Yaskawa INFORM job: A_ROOF_UPPER_0614_2_PAINT_50.JBI

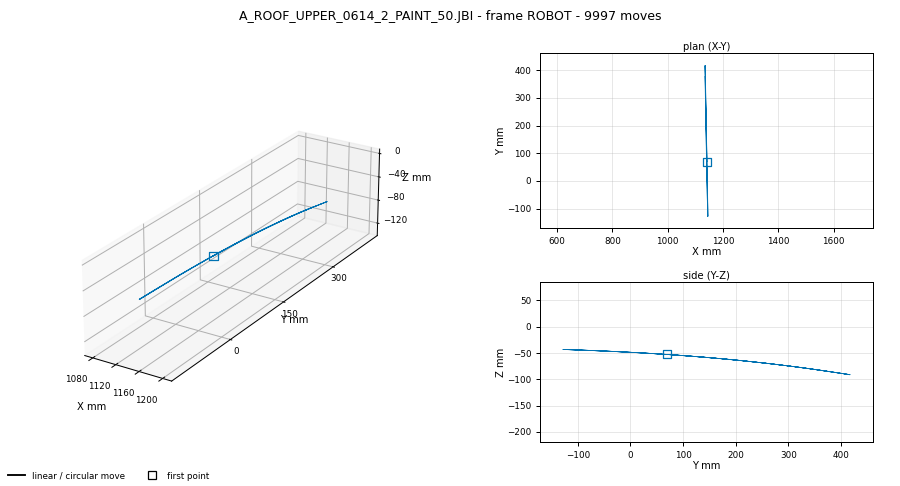
[picture p0: tool path of A_ROOF_UPPER_0614_2_PAINT_50.JBI in frame ROBOT, 9997 of 9997 moves have a stored position in this frame; points joined in program order, loops and branches not executed]
/JOB
//NAME A_ROOF_UPPER_0614_2_PAINT50
//POS
///NPOS 9997,0,0,0,0,0
///TOOL 1
///USER 0
///POSTYPE ROBOT
///RECTAN
///RCONF 1,0,0,0,0,0,0,0,0,0,0,0,0,0,0,0,0,0,0,0,0,0,0,0
C00000=1142.338,69.262,-52.629,-179.610,6.508,149.074
C00001=1142.333,69.511,-52.645,-179.607,6.509,149.073
C00002=1142.328,69.760,-52.662,-179.604,6.511,149.073
C00003=1142.323,70.010,-52.679,-179.601,6.511,149.072
C00004=1142.318,70.259,-52.695,-179.599,6.513,149.072
C00005=1142.313,70.509,-52.711,-179.596,6.515,149.071
C00006=1142.309,70.758,-52.728,-179.593,6.515,149.071
C00007=1142.303,71.007,-52.745,-179.591,6.517,149.070
C00008=1142.298,71.257,-52.762,-179.588,6.518,149.070
C00009=1142.294,71.506,-52.778,-179.585,6.519,149.069
C00010=1142.288,71.755,-52.795,-179.582,6.521,149.069
C00011=1142.284,72.005,-52.812,-179.580,6.522,149.068
C00012=1142.279,72.254,-52.828,-179.578,6.523,149.068
C00013=1142.273,72.503,-52.845,-179.574,6.524,149.067
C00014=1142.269,72.753,-52.862,-179.572,6.526,149.067
C00015=1142.264,73.003,-52.879,-179.569,6.527,149.066
C00016=1142.259,73.251,-52.896,-179.566,6.528,149.066
C00017=1142.254,73.501,-52.912,-179.563,6.530,149.065
C00018=1142.249,73.751,-52.930,-179.561,6.531,149.065
C00019=1142.244,74.000,-52.946,-179.559,6.532,149.064
C00020=1142.239,74.249,-52.962,-179.555,6.534,149.064
C00021=1142.234,74.499,-52.980,-179.553,6.535,149.063
C00022=1142.230,74.748,-52.996,-179.550,6.536,149.063
C00023=1142.224,74.997,-53.013,-179.548,6.538,149.062
C00024=1142.219,75.247,-53.030,-179.544,6.539,149.062
C00025=1142.214,75.497,-53.047,-179.542,6.540,149.061
C00026=1142.209,75.745,-53.064,-179.540,6.542,149.061
C00027=1142.205,75.995,-53.080,-179.537,6.543,149.060
C00028=1142.199,76.245,-53.097,-179.534,6.544,149.060
C00029=1142.195,76.494,-53.114,-179.531,6.546,149.059
C00030=1142.189,76.743,-53.132,-179.529,6.547,149.059
C00031=1142.185,76.992,-53.148,-179.526,6.548,149.058
C00032=1142.180,77.242,-53.166,-179.523,6.549,149.058
C00033=1142.175,77.491,-53.182,-179.521,6.551,149.057
C00034=1142.169,77.741,-53.199,-179.518,6.553,149.057
C00035=1142.165,77.990,-53.216,-179.515,6.553,149.056
C00036=1142.160,78.240,-53.233,-179.513,6.555,149.056
C00037=1142.155,78.489,-53.251,-179.510,6.556,149.055
C00038=1142.150,78.738,-53.268,-179.507,6.558,149.055
C00039=1142.145,78.987,-53.284,-179.504,6.559,149.054
C00040=1142.140,79.256,-53.303,-179.502,6.560,149.054
C00041=1142.134,79.525,-53.322,-179.499,6.562,149.054
C00042=1142.129,79.793,-53.339,-179.496,6.563,149.053
C00043=1142.124,80.061,-53.359,-179.493,6.565,149.052
C00044=1142.120,80.311,-53.375,-179.490,6.566,149.052
C00045=1142.114,80.560,-53.392,-179.487,6.568,149.051
C00046=1142.109,80.810,-53.410,-179.485,6.569,149.051
C00047=1142.104,81.058,-53.427,-179.482,6.570,149.051
C00048=1142.099,81.308,-53.444,-179.479,6.572,149.050
C00049=1142.095,81.558,-53.461,-179.476,6.573,149.049
C00050=1142.090,81.807,-53.479,-179.474,6.574,149.049
C00051=1142.084,82.056,-53.496,-179.471,6.576,149.049
C00052=1142.079,82.305,-53.512,-179.468,6.578,149.048
C00053=1142.075,82.555,-53.530,-179.465,6.579,149.048
C00054=1142.069,82.804,-53.548,-179.463,6.580,149.047
C00055=1142.065,83.054,-53.564,-179.460,6.581,149.047
C00056=1142.060,83.303,-53.582,-179.458,6.583,149.046
C00057=1142.055,83.553,-53.599,-179.454,6.584,149.046
C00058=1142.050,83.801,-53.617,-179.452,6.585,149.045
C00059=1142.045,84.051,-53.634,-179.450,6.587,149.045
C00060=1142.040,84.300,-53.652,-179.447,6.589,149.044
C00061=1142.035,84.549,-53.668,-179.444,6.590,149.044
C00062=1142.030,84.799,-53.686,-179.441,6.591,149.043
C00063=1142.025,85.048,-53.704,-179.439,6.592,149.043
C00064=1142.021,85.298,-53.720,-179.436,6.594,149.042
C00065=1142.016,85.547,-53.738,-179.433,6.596,149.042
C00066=1142.011,85.797,-53.756,-179.430,6.597,149.041
C00067=1142.006,86.046,-53.773,-179.428,6.598,149.041
C00068=1142.001,86.296,-53.790,-179.425,6.599,149.040
C00069=1141.996,86.544,-53.808,-179.422,6.601,149.040
C00070=1141.990,86.794,-53.825,-179.419,6.602,149.039
C00071=1141.986,87.043,-53.843,-179.417,6.603,149.039
C00072=1141.981,87.292,-53.861,-179.414,6.605,149.039
C00073=1141.976,87.542,-53.878,-179.411,6.607,149.038
C00074=1141.971,87.791,-53.896,-179.409,6.608,149.038
C00075=1141.966,88.041,-53.913,-179.406,6.610,149.037
C00076=1141.962,88.289,-53.930,-179.403,6.611,149.037
C00077=1141.957,88.539,-53.948,-179.401,6.612,149.036
C00078=1141.952,88.788,-53.966,-179.398,6.614,149.036
C00079=1141.947,89.038,-53.984,-179.395,6.615,149.035
C00080=1141.942,89.287,-54.001,-179.392,6.617,149.035
C00081=1141.937,89.537,-54.019,-179.390,6.618,149.034
C00082=1141.932,89.785,-54.036,-179.387,6.619,149.034
C00083=1141.927,90.035,-54.054,-179.384,6.621,149.033
C00084=1141.922,90.284,-54.072,-179.381,6.622,149.033
C00085=1141.917,90.534,-54.089,-179.378,6.624,149.032
C00086=1141.913,90.783,-54.107,-179.376,6.626,149.032
C00087=1141.907,91.033,-54.125,-179.373,6.627,149.032
C00088=1141.902,91.282,-54.143,-179.371,6.628,149.031
C00089=1141.898,91.531,-54.160,-179.368,6.630,149.030
C00090=1141.893,91.780,-54.178,-179.365,6.631,149.030
C00091=1141.888,92.030,-54.195,-179.362,6.633,149.030
C00092=1141.883,92.279,-54.213,-179.360,6.634,149.029
C00093=1141.878,92.528,-54.231,-179.357,6.635,149.029
C00094=1141.873,92.777,-54.249,-179.354,6.637,149.028
C00095=1141.868,93.027,-54.267,-179.351,6.638,149.028
C00096=1141.863,93.276,-54.285,-179.348,6.640,149.027
C00097=1141.858,93.525,-54.303,-179.346,6.642,149.027
C00098=1141.854,93.775,-54.321,-179.344,6.643,149.026
C00099=1141.849,94.024,-54.339,-179.340,6.644,149.026
C00100=1141.844,94.273,-54.357,-179.338,6.646,149.025
C00101=1141.839,94.523,-54.374,-179.335,6.647,149.025
C00102=1141.834,94.772,-54.392,-179.332,6.649,149.025
C00103=1141.829,95.022,-54.410,-179.329,6.651,149.024
C00104=1141.824,95.271,-54.428,-179.327,6.652,149.024
C00105=1141.819,95.520,-54.446,-179.324,6.653,149.023
C00106=1141.814,95.769,-54.464,-179.321,6.654,149.023
C00107=1141.809,96.018,-54.482,-179.319,6.656,149.022
C00108=1141.805,96.268,-54.500,-179.316,6.658,149.022
C00109=1141.800,96.517,-54.518,-179.313,6.659,149.021
C00110=1141.795,96.767,-54.536,-179.310,6.661,149.021
C00111=1141.790,97.016,-54.554,-179.307,6.662,149.020
C00112=1141.786,97.265,-54.572,-179.305,6.663,149.020
C00113=1141.781,97.514,-54.590,-179.302,6.665,149.020
C00114=1141.776,97.763,-54.608,-179.300,6.667,149.019
C00115=1141.771,98.012,-54.626,-179.297,6.668,149.019
C00116=1141.766,98.262,-54.645,-179.294,6.670,149.018
C00117=1141.762,98.511,-54.662,-179.291,6.671,149.018
C00118=1141.756,98.761,-54.681,-179.288,6.673,149.017
C00119=1141.751,99.010,-54.699,-179.285,6.675,149.017
C00120=1141.746,99.259,-54.717,-179.283,6.676,149.016
C00121=1141.741,99.509,-54.735,-179.281,6.677,149.016
C00122=1141.737,99.758,-54.753,-179.278,6.679,149.016
C00123=1141.732,100.008,-54.771,-179.275,6.680,149.015
C00124=1141.727,100.257,-54.789,-179.272,6.682,149.014
C00125=1141.722,100.506,-54.807,-179.269,6.684,149.014
C00126=1141.717,100.755,-54.827,-179.266,6.685,149.014
C00127=1141.712,101.005,-54.845,-179.264,6.687,149.013
C00128=1141.708,101.254,-54.863,-179.261,6.689,149.013
C00129=1141.703,101.503,-54.881,-179.258,6.689,149.012
C00130=1141.698,101.752,-54.899,-179.256,6.691,149.012
C00131=1141.692,102.002,-54.917,-179.253,6.692,149.011
C00132=1141.688,102.251,-54.936,-179.250,6.694,149.011
C00133=1141.683,102.500,-54.954,-179.247,6.696,149.011
C00134=1141.678,102.749,-54.972,-179.245,6.698,149.010
C00135=1141.673,102.998,-54.990,-179.242,6.699,149.010
C00136=1141.669,103.248,-55.010,-179.239,6.701,149.009
C00137=1141.664,103.497,-55.028,-179.236,6.702,149.009
C00138=1141.659,103.746,-55.046,-179.233,6.704,149.008
C00139=1141.654,103.996,-55.064,-179.231,6.706,149.008
C00140=1141.649,104.245,-55.084,-179.228,6.706,149.007
C00141=1141.644,104.494,-55.102,-179.226,6.708,149.007
C00142=1141.639,104.743,-55.120,-179.223,6.710,149.007
C00143=1141.635,104.993,-55.139,-179.220,6.711,149.006
C00144=1141.629,105.261,-55.159,-179.217,6.713,149.006
C00145=1141.624,105.530,-55.178,-179.214,6.715,149.005
C00146=1141.619,105.798,-55.198,-179.211,6.717,149.005
C00147=1141.614,106.066,-55.218,-179.208,6.718,149.004
C00148=1141.609,106.316,-55.237,-179.205,6.720,149.004
C00149=1141.604,106.565,-55.255,-179.202,6.722,149.003
C00150=1141.599,106.814,-55.274,-179.199,6.723,149.003
C00151=1141.594,107.064,-55.293,-179.197,6.725,149.002
C00152=1141.590,107.312,-55.312,-179.194,6.727,149.002
C00153=1141.584,107.562,-55.330,-179.192,6.728,149.002
C00154=1141.580,107.812,-55.348,-179.189,6.729,149.001
C00155=1141.575,108.060,-55.367,-179.186,6.731,149.001
C00156=1141.569,108.310,-55.386,-179.183,6.732,149.000
C00157=1141.565,108.559,-55.405,-179.180,6.734,149.000
C00158=1141.560,108.808,-55.423,-179.178,6.736,148.999
C00159=1141.555,109.057,-55.442,-179.175,6.737,148.999
C00160=1141.551,109.307,-55.460,-179.172,6.739,148.999
C00161=1141.545,109.556,-55.480,-179.170,6.741,148.998
C00162=1141.541,109.806,-55.498,-179.167,6.742,148.998
C00163=1141.536,110.055,-55.517,-179.164,6.744,148.997
C00164=1141.531,110.304,-55.535,-179.161,6.745,148.997
C00165=1141.527,110.553,-55.554,-179.158,6.747,148.996
C00166=1141.522,110.802,-55.574,-179.155,6.749,148.996
C00167=1141.517,111.052,-55.592,-179.153,6.750,148.995
C00168=1141.512,111.301,-55.611,-179.150,6.752,148.995
C00169=1141.507,111.550,-55.629,-179.147,6.754,148.995
C00170=1141.502,111.799,-55.649,-179.145,6.755,148.994
C00171=1141.498,112.048,-55.668,-179.142,6.757,148.994
C00172=1141.493,112.298,-55.687,-179.139,6.759,148.993
C00173=1141.488,112.547,-55.705,-179.136,6.760,148.993
C00174=1141.482,112.796,-55.724,-179.133,6.762,148.992
C00175=1141.478,113.046,-55.743,-179.130,6.764,148.992
C00176=1141.473,113.294,-55.762,-179.128,6.765,148.992
C00177=1141.468,113.544,-55.782,-179.125,6.767,148.991
C00178=1141.463,113.793,-55.800,-179.122,6.769,148.991
C00179=1141.459,114.043,-55.819,-179.119,6.770,148.990
C00180=1141.454,114.291,-55.838,-179.117,6.772,148.990
C00181=1141.449,114.541,-55.857,-179.114,6.774,148.990
C00182=1141.444,114.790,-55.876,-179.111,6.775,148.989
C00183=1141.440,115.039,-55.895,-179.109,6.777,148.989
C00184=1141.434,115.288,-55.915,-179.106,6.779,148.988
C00185=1141.430,115.538,-55.933,-179.103,6.780,148.988
C00186=1141.425,115.787,-55.952,-179.100,6.782,148.987
C00187=1141.420,116.037,-55.972,-179.097,6.783,148.987
C00188=1141.415,116.285,-55.991,-179.094,6.785,148.986
C00189=1141.410,116.535,-56.010,-179.092,6.787,148.986
C00190=1141.406,116.783,-56.029,-179.089,6.788,148.986
C00191=1141.401,117.034,-56.048,-179.086,6.790,148.985
C00192=1141.395,117.282,-56.067,-179.084,6.792,148.985
C00193=1141.391,117.532,-56.086,-179.081,6.794,148.984
C00194=1141.386,117.781,-56.106,-179.078,6.795,148.984
C00195=1141.381,118.030,-56.125,-179.075,6.797,148.984
C00196=1141.376,118.279,-56.145,-179.073,6.799,148.983
C00197=1141.372,118.528,-56.164,-179.070,6.800,148.983
C00198=1141.367,118.777,-56.183,-179.067,6.802,148.982
C00199=1141.362,119.027,-56.203,-179.064,6.804,148.982
C00200=1141.357,119.276,-56.221,-179.062,6.805,148.982
C00201=1141.352,119.525,-56.240,-179.059,6.807,148.981
C00202=1141.348,119.775,-56.260,-179.056,6.808,148.981
C00203=1141.342,120.024,-56.279,-179.053,6.810,148.980
C00204=1141.338,120.273,-56.298,-179.050,6.812,148.980
C00205=1141.333,120.522,-56.318,-179.048,6.813,148.979
C00206=1141.328,120.772,-56.337,-179.045,6.815,148.979
C00207=1141.323,121.021,-56.357,-179.042,6.817,148.979
C00208=1141.319,121.270,-56.376,-179.039,6.819,148.978
C00209=1141.314,121.519,-56.396,-179.037,6.820,148.978
C00210=1141.309,121.767,-56.415,-179.034,6.822,148.977
C00211=1141.304,122.017,-56.435,-179.031,6.824,148.977
C00212=1141.299,122.267,-56.455,-179.028,6.826,148.977
C00213=1141.295,122.515,-56.473,-179.025,6.828,148.976
C00214=1141.290,122.765,-56.493,-179.023,6.830,148.976
C00215=1141.285,123.014,-56.513,-179.020,6.831,148.975
C00216=1141.280,123.263,-56.532,-179.017,6.833,148.975
C00217=1141.275,123.513,-56.551,-179.014,6.835,148.975
C00218=1141.270,123.762,-56.571,-179.012,6.836,148.974
C00219=1141.266,124.010,-56.591,-179.009,6.838,148.974
C00220=1141.262,124.260,-56.610,-179.006,6.840,148.973
C00221=1141.256,124.509,-56.629,-179.003,6.841,148.973
C00222=1141.251,124.758,-56.649,-179.001,6.843,148.973
C00223=1141.247,125.008,-56.669,-178.998,6.845,148.972
C00224=1141.242,125.257,-56.689,-178.995,6.846,148.972
C00225=1141.237,125.506,-56.708,-178.992,6.849,148.971
C00226=1141.232,125.755,-56.728,-178.989,6.851,148.971
C00227=1141.227,126.005,-56.748,-178.987,6.852,148.971
C00228=1141.223,126.253,-56.767,-178.984,6.854,148.970
C00229=1141.218,126.502,-56.787,-178.981,6.856,148.970
C00230=1141.214,126.752,-56.807,-178.978,6.857,148.969
C00231=1141.208,127.001,-56.826,-178.976,6.859,148.969
C00232=1141.204,127.250,-56.846,-178.973,6.861,148.969
C00233=1141.199,127.499,-56.866,-178.970,6.863,148.968
C00234=1141.194,127.749,-56.885,-178.967,6.864,148.968
C00235=1141.189,127.997,-56.905,-178.965,6.866,148.967
C00236=1141.185,128.247,-56.925,-178.961,6.868,148.967
C00237=1141.180,128.496,-56.945,-178.959,6.870,148.967
C00238=1141.175,128.745,-56.965,-178.956,6.872,148.966
C00239=1141.170,128.994,-56.984,-178.953,6.873,148.966
C00240=1141.166,129.243,-57.005,-178.951,6.875,148.965
C00241=1141.161,129.493,-57.024,-178.948,6.877,148.965
C00242=1141.156,129.742,-57.044,-178.945,6.879,148.965
C00243=1141.151,129.990,-57.064,-178.942,6.880,148.964
C00244=1141.146,130.240,-57.084,-178.940,6.882,148.964
C00245=1141.141,130.489,-57.105,-178.936,6.884,148.963
C00246=1141.136,130.739,-57.124,-178.934,6.886,148.963
C00247=1141.132,130.988,-57.145,-178.931,6.888,148.963
C00248=1141.127,131.256,-57.166,-178.928,6.890,148.962
C00249=1141.121,131.525,-57.188,-178.925,6.892,148.962
C00250=1141.117,131.793,-57.209,-178.922,6.893,148.961
C00251=1141.111,132.061,-57.230,-178.919,6.895,148.961
C00252=1141.106,132.311,-57.251,-178.916,6.897,148.960
C00253=1141.101,132.560,-57.271,-178.913,6.899,148.960
C00254=1141.097,132.809,-57.291,-178.910,6.901,148.960
C00255=1141.092,133.059,-57.311,-178.908,6.903,148.959
C00256=1141.088,133.308,-57.331,-178.905,6.904,148.959
C00257=1141.082,133.556,-57.350,-178.903,6.906,148.959
C00258=1141.077,133.806,-57.371,-178.900,6.908,148.958
C00259=1141.073,134.055,-57.392,-178.897,6.910,148.958
C00260=1141.068,134.304,-57.411,-178.894,6.912,148.958
C00261=1141.064,134.553,-57.432,-178.891,6.914,148.957
C00262=1141.059,134.802,-57.452,-178.888,6.916,148.957
C00263=1141.054,135.052,-57.472,-178.886,6.917,148.956
C00264=1141.049,135.301,-57.493,-178.883,6.919,148.956
C00265=1141.044,135.549,-57.513,-178.880,6.921,148.956
C00266=1141.040,135.799,-57.532,-178.877,6.923,148.955
C00267=1141.035,136.048,-57.553,-178.874,6.925,148.955
C00268=1141.030,136.297,-57.574,-178.871,6.927,148.954
C00269=1141.025,136.547,-57.593,-178.869,6.929,148.954
C00270=1141.021,136.795,-57.614,-178.866,6.930,148.954
C00271=1141.016,137.044,-57.634,-178.863,6.932,148.953
C00272=1141.011,137.294,-57.655,-178.860,6.934,148.953
C00273=1141.006,137.543,-57.675,-178.857,6.936,148.952
C00274=1141.002,137.792,-57.695,-178.855,6.938,148.952
C00275=1140.997,138.041,-57.716,-178.852,6.940,148.952
C00276=1140.992,138.290,-57.736,-178.850,6.942,148.952
C00277=1140.988,138.539,-57.757,-178.846,6.944,148.951
C00278=1140.982,138.788,-57.777,-178.844,6.946,148.951
C00279=1140.977,139.037,-57.797,-178.841,6.948,148.950
C00280=1140.973,139.286,-57.817,-178.838,6.949,148.950
C00281=1140.968,139.536,-57.838,-178.835,6.951,148.950
C00282=1140.963,139.785,-57.859,-178.833,6.953,148.949
C00283=1140.959,140.034,-57.879,-178.829,6.955,148.949
C00284=1140.954,140.283,-57.900,-178.827,6.957,148.948
C00285=1140.949,140.532,-57.921,-178.824,6.959,148.948
C00286=1140.945,140.781,-57.941,-178.821,6.960,148.948
C00287=1140.940,141.030,-57.962,-178.819,6.962,148.947
C00288=1140.935,141.279,-57.982,-178.816,6.965,148.947
C00289=1140.930,141.528,-58.003,-178.813,6.967,148.947
C00290=1140.926,141.777,-58.024,-178.810,6.968,148.946
C00291=1140.921,142.026,-58.044,-178.808,6.970,148.946
C00292=1140.916,142.275,-58.065,-178.804,6.972,148.946
C00293=1140.912,142.524,-58.085,-178.802,6.974,148.945
C00294=1140.907,142.774,-58.107,-178.799,6.976,148.945
C00295=1140.903,143.023,-58.127,-178.796,6.978,148.944
C00296=1140.897,143.272,-58.148,-178.793,6.979,148.944
C00297=1140.893,143.521,-58.168,-178.790,6.982,148.944
C00298=1140.888,143.771,-58.189,-178.788,6.984,148.943
C00299=1140.883,144.020,-58.210,-178.785,6.986,148.943
C00300=1140.879,144.269,-58.230,-178.782,6.987,148.943
C00301=1140.874,144.518,-58.251,-178.779,6.990,148.942
C00302=1140.869,144.767,-58.271,-178.776,6.991,148.942
C00303=1140.864,145.016,-58.292,-178.774,6.993,148.942
C00304=1140.859,145.265,-58.313,-178.771,6.995,148.941
C00305=1140.855,145.514,-58.334,-178.768,6.997,148.941
C00306=1140.850,145.763,-58.355,-178.765,6.999,148.940
C00307=1140.845,146.012,-58.376,-178.763,7.001,148.940
C00308=1140.841,146.262,-58.397,-178.760,7.003,148.940
C00309=1140.836,146.511,-58.417,-178.757,7.005,148.939
C00310=1140.831,146.759,-58.439,-178.754,7.007,148.939
C00311=1140.827,147.008,-58.460,-178.751,7.009,148.939
C00312=1140.822,147.258,-58.480,-178.749,7.011,148.938
C00313=1140.817,147.507,-58.501,-178.746,7.012,148.938
C00314=1140.812,147.756,-58.522,-178.743,7.015,148.938
C00315=1140.807,148.004,-58.544,-178.740,7.017,148.937
C00316=1140.803,148.254,-58.565,-178.738,7.019,148.937
C00317=1140.798,148.503,-58.585,-178.734,7.021,148.937
C00318=1140.793,148.752,-58.607,-178.732,7.023,148.936
C00319=1140.789,149.001,-58.627,-178.729,7.024,148.936
C00320=1140.784,149.250,-58.648,-178.726,7.026,148.935
C00321=1140.779,149.499,-58.670,-178.723,7.029,148.935
C00322=1140.775,149.749,-58.691,-178.721,7.031,148.935
C00323=1140.770,149.998,-58.712,-178.718,7.032,148.935
C00324=1140.765,150.246,-58.733,-178.715,7.034,148.934
C00325=1140.760,150.496,-58.754,-178.712,7.037,148.934
C00326=1140.755,150.745,-58.775,-178.709,7.038,148.933
C00327=1140.751,150.994,-58.797,-178.707,7.040,148.933
C00328=1140.746,151.243,-58.818,-178.704,7.043,148.933
C00329=1140.742,151.492,-58.839,-178.701,7.045,148.933
C00330=1140.737,151.741,-58.860,-178.698,7.046,148.932
C00331=1140.732,151.989,-58.881,-178.695,7.048,148.932
C00332=1140.727,152.239,-58.903,-178.692,7.051,148.931
C00333=1140.723,152.488,-58.924,-178.690,7.053,148.931
C00334=1140.718,152.737,-58.945,-178.687,7.054,148.931
C00335=1140.713,152.986,-58.966,-178.684,7.057,148.930
C00336=1140.708,153.236,-58.988,-178.681,7.059,148.930
C00337=1140.704,153.484,-59.009,-178.678,7.060,148.930
C00338=1140.699,153.733,-59.030,-178.675,7.063,148.929
C00339=1140.694,153.982,-59.052,-178.673,7.065,148.929
C00340=1140.690,154.232,-59.073,-178.670,7.067,148.929
C00341=1140.685,154.480,-59.095,-178.668,7.068,148.928
C00342=1140.680,154.730,-59.116,-178.664,7.071,148.928
C00343=1140.675,154.978,-59.137,-178.662,7.073,148.928
C00344=1140.671,155.227,-59.159,-178.659,7.075,148.928
C00345=1140.666,155.477,-59.180,-178.656,7.077,148.927
C00346=1140.661,155.725,-59.201,-178.653,7.079,148.927
C00347=1140.657,155.975,-59.223,-178.651,7.081,148.926
C00348=1140.652,156.224,-59.244,-178.647,7.083,148.926
C00349=1140.647,156.472,-59.266,-178.645,7.085,148.926
C00350=1140.643,156.722,-59.288,-178.642,7.087,148.925
C00351=1140.637,156.971,-59.309,-178.639,7.090,148.925
C00352=1140.633,157.240,-59.332,-178.636,7.091,148.925
C00353=1140.627,157.509,-59.356,-178.633,7.094,148.924
C00354=1140.623,157.778,-59.379,-178.630,7.095,148.924
C00355=1140.618,158.047,-59.403,-178.627,7.098,148.924
C00356=1140.612,158.296,-59.424,-178.625,7.100,148.923
C00357=1140.608,158.545,-59.445,-178.621,7.103,148.923
C00358=1140.604,158.794,-59.467,-178.619,7.104,148.923
C00359=1140.599,159.042,-59.488,-178.616,7.106,148.922
C00360=1140.594,159.291,-59.509,-178.613,7.109,148.922
C00361=1140.590,159.541,-59.531,-178.611,7.111,148.922
C00362=1140.585,159.789,-59.553,-178.607,7.113,148.921
C00363=1140.581,160.039,-59.575,-178.605,7.115,148.921
C00364=1140.576,160.287,-59.597,-178.602,7.117,148.921
C00365=1140.571,160.536,-59.619,-178.599,7.119,148.921
C00366=1140.567,160.785,-59.641,-178.596,7.121,148.920
C00367=1140.561,161.035,-59.662,-178.594,7.123,148.920
C00368=1140.556,161.284,-59.684,-178.590,7.125,148.919
C00369=1140.551,161.533,-59.706,-178.588,7.127,148.919
C00370=1140.547,161.782,-59.728,-178.585,7.129,148.919
C00371=1140.542,162.031,-59.750,-178.582,7.132,148.919
C00372=1140.537,162.280,-59.771,-178.579,7.133,148.918
C00373=1140.533,162.529,-59.793,-178.577,7.136,148.918
C00374=1140.528,162.778,-59.815,-178.574,7.138,148.918
C00375=1140.524,163.027,-59.837,-178.571,7.140,148.917
C00376=1140.519,163.276,-59.859,-178.568,7.142,148.917
C00377=1140.515,163.525,-59.881,-178.566,7.144,148.917
C00378=1140.510,163.774,-59.903,-178.563,7.146,148.916
C00379=1140.506,164.023,-59.925,-178.560,7.149,148.916
C00380=1140.500,164.272,-59.947,-178.557,7.150,148.916
C00381=1140.496,164.521,-59.969,-178.554,7.153,148.916
C00382=1140.491,164.770,-59.991,-178.551,7.155,148.915
C00383=1140.487,165.019,-60.013,-178.549,7.157,148.915
C00384=1140.482,165.268,-60.034,-178.545,7.159,148.914
C00385=1140.478,165.517,-60.057,-178.543,7.161,148.914
C00386=1140.472,165.765,-60.079,-178.540,7.164,148.914
C00387=1140.468,166.015,-60.101,-178.537,7.166,148.914
C00388=1140.463,166.263,-60.123,-178.535,7.168,148.913
C00389=1140.459,166.513,-60.145,-178.532,7.170,148.913
C00390=1140.454,166.761,-60.167,-178.529,7.172,148.913
C00391=1140.449,167.011,-60.189,-178.526,7.174,148.912
C00392=1140.445,167.259,-60.212,-178.523,7.176,148.912
C00393=1140.440,167.508,-60.234,-178.521,7.178,148.912
C00394=1140.435,167.757,-60.256,-178.517,7.181,148.911
C00395=1140.430,168.007,-60.278,-178.515,7.183,148.911
C00396=1140.426,168.255,-60.301,-178.512,7.185,148.911
C00397=1140.422,168.504,-60.323,-178.509,7.187,148.911
C00398=1140.417,168.754,-60.345,-178.506,7.190,148.910
C00399=1140.412,169.002,-60.367,-178.504,7.192,148.910
C00400=1140.408,169.251,-60.390,-178.501,7.193,148.910
C00401=1140.403,169.500,-60.411,-178.498,7.196,148.909
C00402=1140.398,169.749,-60.434,-178.495,7.198,148.909
C00403=1140.394,169.998,-60.457,-178.492,7.200,148.909
C00404=1140.389,170.247,-60.479,-178.489,7.202,148.908
C00405=1140.384,170.496,-60.501,-178.487,7.205,148.908
C00406=1140.379,170.744,-60.524,-178.484,7.207,148.908
C00407=1140.374,170.994,-60.546,-178.481,7.209,148.908
C00408=1140.370,171.243,-60.568,-178.478,7.211,148.907
C00409=1140.366,171.491,-60.591,-178.476,7.213,148.907
C00410=1140.361,171.741,-60.613,-178.472,7.216,148.907
C00411=1140.356,171.989,-60.636,-178.470,7.218,148.907
C00412=1140.352,172.238,-60.658,-178.467,7.220,148.906
C00413=1140.347,172.488,-60.680,-178.464,7.222,148.906
C00414=1140.342,172.736,-60.703,-178.461,7.225,148.906
C00415=1140.337,172.986,-60.725,-178.459,7.227,148.905
C00416=1140.333,173.235,-60.748,-178.455,7.229,148.905
C00417=1140.328,173.483,-60.770,-178.453,7.231,148.905
C00418=1140.324,173.732,-60.793,-178.450,7.233,148.905
C00419=1140.319,173.982,-60.816,-178.447,7.235,148.904
C00420=1140.314,174.230,-60.838,-178.445,7.238,148.904
C00421=1140.310,174.479,-60.861,-178.442,7.240,148.904
C00422=1140.305,174.728,-60.884,-178.439,7.242,148.904
C00423=1140.301,174.977,-60.906,-178.436,7.245,148.903
C00424=1140.296,175.226,-60.929,-178.433,7.246,148.903
C00425=1140.292,175.475,-60.952,-178.430,7.249,148.903
C00426=1140.287,175.724,-60.974,-178.428,7.251,148.902
C00427=1140.282,175.972,-60.997,-178.425,7.254,148.902
C00428=1140.277,176.221,-61.020,-178.422,7.256,148.902
C00429=1140.272,176.471,-61.043,-178.419,7.258,148.901
C00430=1140.268,176.720,-61.065,-178.416,7.260,148.901
C00431=1140.263,176.968,-61.088,-178.413,7.263,148.901
C00432=1140.259,177.217,-61.110,-178.411,7.265,148.901
C00433=1140.254,177.466,-61.134,-178.408,7.267,148.900
C00434=1140.250,177.715,-61.156,-178.405,7.269,148.900
C00435=1140.245,177.964,-61.179,-178.402,7.272,148.900
C00436=1140.240,178.213,-61.202,-178.400,7.274,148.900
C00437=1140.236,178.462,-61.225,-178.396,7.276,148.899
C00438=1140.231,178.711,-61.248,-178.394,7.278,148.899
C00439=1140.226,178.960,-61.270,-178.391,7.281,148.899
C00440=1140.222,179.209,-61.293,-178.388,7.283,148.898
C00441=1140.217,179.458,-61.317,-178.385,7.286,148.898
C00442=1140.213,179.706,-61.339,-178.383,7.287,148.898
C00443=1140.208,179.955,-61.363,-178.380,7.290,148.898
C00444=1140.204,180.204,-61.386,-178.377,7.292,148.897
C00445=1140.199,180.453,-61.408,-178.374,7.294,148.897
C00446=1140.194,180.702,-61.431,-178.372,7.297,148.897
C00447=1140.189,180.951,-61.455,-178.368,7.299,148.897
C00448=1140.185,181.200,-61.477,-178.366,7.301,148.896
C00449=1140.181,181.449,-61.501,-178.363,7.304,148.896
C00450=1140.176,181.698,-61.524,-178.360,7.305,148.896
C00451=1140.171,181.946,-61.546,-178.357,7.308,148.896
C00452=1140.167,182.195,-61.570,-178.355,7.310,148.895
C00453=1140.162,182.444,-61.593,-178.352,7.313,148.895
C00454=1140.157,182.693,-61.616,-178.349,7.315,148.895
C00455=1140.153,182.942,-61.639,-178.346,7.318,148.895
C00456=1140.148,183.211,-61.664,-178.343,7.320,148.894
C00457=1140.143,183.481,-61.689,-178.340,7.323,148.894
C00458=1140.137,183.751,-61.714,-178.336,7.325,148.894
C00459=1140.133,184.020,-61.739,-178.334,7.327,148.893
C00460=1140.128,184.269,-61.762,-178.331,7.330,148.893
C00461=1140.124,184.518,-61.786,-178.328,7.333,148.893
C00462=1140.119,184.767,-61.810,-178.325,7.334,148.893
C00463=1140.114,185.016,-61.833,-178.323,7.337,148.893
C00464=1140.110,185.265,-61.856,-178.320,7.339,148.892
C00465=1140.106,185.514,-61.879,-178.317,7.342,148.892
C00466=1140.101,185.763,-61.902,-178.314,7.344,148.892
C00467=1140.096,186.012,-61.926,-178.311,7.346,148.891
C00468=1140.091,186.261,-61.949,-178.309,7.348,148.891
C00469=1140.087,186.510,-61.972,-178.306,7.351,148.891
C00470=1140.082,186.758,-61.997,-178.303,7.354,148.891
C00471=1140.078,187.007,-62.020,-178.300,7.355,148.890
C00472=1140.074,187.256,-62.043,-178.297,7.358,148.890
C00473=1140.069,187.505,-62.066,-178.295,7.360,148.890
C00474=1140.064,187.753,-62.089,-178.292,7.363,148.890
C00475=1140.059,188.002,-62.113,-178.289,7.365,148.889
C00476=1140.055,188.251,-62.136,-178.286,7.368,148.889
C00477=1140.050,188.500,-62.160,-178.283,7.370,148.889
C00478=1140.045,188.749,-62.183,-178.281,7.372,148.889
C00479=1140.041,188.997,-62.207,-178.277,7.375,148.889
C00480=1140.036,189.246,-62.231,-178.275,7.377,148.888
C00481=1140.031,189.495,-62.254,-178.272,7.379,148.888
C00482=1140.027,189.744,-62.277,-178.269,7.382,148.888
C00483=1140.022,189.993,-62.301,-178.266,7.384,148.888
C00484=1140.018,190.242,-62.325,-178.264,7.387,148.887
C00485=1140.013,190.491,-62.348,-178.261,7.389,148.887
C00486=1140.009,190.739,-62.372,-178.258,7.392,148.887
C00487=1140.004,190.989,-62.396,-178.255,7.394,148.887
C00488=1140.000,191.237,-62.420,-178.253,7.396,148.886
C00489=1139.995,191.486,-62.443,-178.249,7.399,148.886
C00490=1139.991,191.736,-62.467,-178.247,7.401,148.886
C00491=1139.986,191.984,-62.491,-178.244,7.403,148.886
C00492=1139.982,192.233,-62.514,-178.241,7.406,148.886
C00493=1139.977,192.481,-62.538,-178.238,7.408,148.885
C00494=1139.972,192.731,-62.562,-178.236,7.411,148.885
C00495=1139.967,192.979,-62.586,-178.233,7.413,148.885
C00496=1139.963,193.228,-62.610,-178.230,7.416,148.885
C00497=1139.958,193.477,-62.634,-178.227,7.418,148.884
C00498=1139.954,193.726,-62.657,-178.225,7.420,148.884
C00499=1139.949,193.974,-62.681,-178.221,7.423,148.884
C00500=1139.945,194.224,-62.705,-178.218,7.426,148.884
C00501=1139.941,194.472,-62.729,-178.216,7.427,148.883
C00502=1139.935,194.721,-62.753,-178.213,7.430,148.883
C00503=1139.931,194.970,-62.777,-178.211,7.432,148.883
C00504=1139.926,195.219,-62.800,-178.207,7.435,148.883
C00505=1139.922,195.467,-62.824,-178.205,7.438,148.883
C00506=1139.917,195.716,-62.848,-178.202,7.440,148.882
C00507=1139.913,195.965,-62.872,-178.199,7.442,148.882
C00508=1139.908,196.214,-62.897,-178.196,7.445,148.882
C00509=1139.904,196.463,-62.921,-178.194,7.447,148.882
C00510=1139.899,196.712,-62.944,-178.190,7.450,148.881
C00511=1139.895,196.960,-62.968,-178.188,7.452,148.881
C00512=1139.889,197.209,-62.993,-178.185,7.455,148.881
C00513=1139.885,197.458,-63.016,-178.182,7.457,148.881
C00514=1139.881,197.707,-63.041,-178.179,7.460,148.881
C00515=1139.877,197.955,-63.065,-178.177,7.462,148.880
C00516=1139.871,198.204,-63.090,-178.174,7.465,148.880
C00517=1139.867,198.453,-63.113,-178.170,7.467,148.880
C00518=1139.862,198.702,-63.137,-178.168,7.469,148.880
C00519=1139.859,198.951,-63.161,-178.165,7.472,148.880
C00520=1139.853,199.199,-63.186,-178.162,7.475,148.879
C00521=1139.849,199.448,-63.209,-178.160,7.477,148.879
C00522=1139.844,199.697,-63.234,-178.157,7.479,148.879
C00523=1139.840,199.946,-63.259,-178.154,7.482,148.879
C00524=1139.835,200.195,-63.283,-178.152,7.484,148.879
C00525=1139.831,200.443,-63.307,-178.148,7.487,148.878
C00526=1139.826,200.692,-63.331,-178.145,7.490,148.878
C00527=1139.822,200.941,-63.356,-178.143,7.492,148.878
C00528=1139.818,201.189,-63.380,-178.140,7.494,148.878
C00529=1139.812,201.439,-63.404,-178.137,7.497,148.878
C00530=1139.808,201.687,-63.428,-178.134,7.499,148.877
C00531=1139.803,201.936,-63.453,-178.132,7.502,148.877
C00532=1139.799,202.185,-63.477,-178.128,7.505,148.877
C00533=1139.795,202.433,-63.501,-178.126,7.507,148.877
C00534=1139.790,202.683,-63.526,-178.123,7.510,148.877
C00535=1139.786,202.931,-63.550,-178.120,7.512,148.876
C00536=1139.780,203.180,-63.575,-178.117,7.515,148.876
C00537=1139.776,203.428,-63.599,-178.115,7.517,148.876
C00538=1139.772,203.678,-63.624,-178.112,7.520,148.876
C00539=1139.767,203.926,-63.648,-178.109,7.523,148.876
C00540=1139.763,204.175,-63.672,-178.106,7.524,148.875
C00541=1139.758,204.424,-63.697,-178.103,7.527,148.875
C00542=1139.754,204.672,-63.721,-178.101,7.530,148.875
C00543=1139.749,204.920,-63.747,-178.097,7.533,148.875
C00544=1139.745,205.170,-63.771,-178.095,7.535,148.875
C00545=1139.740,205.418,-63.796,-178.092,7.538,148.874
C00546=1139.735,205.667,-63.820,-178.089,7.540,148.874
C00547=1139.731,205.916,-63.845,-178.087,7.542,148.874
C00548=1139.726,206.165,-63.870,-178.084,7.545,148.874
C00549=1139.722,206.414,-63.894,-178.081,7.548,148.874
C00550=1139.717,206.662,-63.919,-178.078,7.551,148.873
C00551=1139.713,206.910,-63.943,-178.076,7.553,148.873
C00552=1139.709,207.160,-63.968,-178.072,7.555,148.873
C00553=1139.703,207.409,-63.993,-178.070,7.558,148.873
C00554=1139.699,207.657,-64.017,-178.067,7.561,148.873
C00555=1139.695,207.906,-64.043,-178.064,7.563,148.872
C00556=1139.690,208.154,-64.067,-178.061,7.566,148.872
C00557=1139.686,208.404,-64.092,-178.059,7.569,148.872
C00558=1139.681,208.652,-64.117,-178.056,7.570,148.872
C00559=1139.677,208.900,-64.142,-178.053,7.573,148.872
C00560=1139.672,209.171,-64.169,-178.050,7.576,148.872
C00561=1139.667,209.442,-64.196,-178.047,7.579,148.871
C00562=1139.662,209.712,-64.223,-178.044,7.582,148.871
C00563=1139.657,209.983,-64.250,-178.040,7.585,148.871
C00564=1139.652,210.232,-64.275,-178.038,7.587,148.871
C00565=1139.648,210.481,-64.300,-178.035,7.590,148.871
C00566=1139.643,210.729,-64.325,-178.032,7.593,148.870
C00567=1139.639,210.979,-64.350,-178.029,7.595,148.870
C00568=1139.635,211.226,-64.374,-178.027,7.598,148.870
C00569=1139.630,211.476,-64.399,-178.024,7.600,148.870
C00570=1139.625,211.724,-64.425,-178.021,7.603,148.870
C00571=1139.621,211.973,-64.450,-178.018,7.606,148.870
C00572=1139.617,212.221,-64.475,-178.016,7.608,148.870
C00573=1139.612,212.471,-64.500,-178.013,7.611,148.869
C00574=1139.607,212.719,-64.525,-178.010,7.613,148.869
C00575=1139.603,212.968,-64.550,-178.007,7.616,148.869
C00576=1139.598,213.216,-64.576,-178.004,7.619,148.869
C00577=1139.594,213.465,-64.600,-178.001,7.621,148.869
C00578=1139.589,213.713,-64.625,-177.999,7.624,148.869
C00579=1139.585,213.963,-64.650,-177.996,7.627,148.868
C00580=1139.580,214.211,-64.676,-177.993,7.630,148.868
C00581=1139.576,214.460,-64.701,-177.990,7.632,148.868
C00582=1139.571,214.708,-64.726,-177.988,7.634,148.868
C00583=1139.567,214.957,-64.751,-177.985,7.637,148.868
C00584=1139.563,215.206,-64.776,-177.982,7.640,148.868
C00585=1139.558,215.455,-64.802,-177.979,7.643,148.867
C00586=1139.554,215.703,-64.827,-177.976,7.646,148.867
C00587=1139.548,215.952,-64.852,-177.974,7.648,148.867
C00588=1139.544,216.201,-64.878,-177.971,7.651,148.867
C00589=1139.539,216.449,-64.903,-177.968,7.653,148.867
C00590=1139.536,216.698,-64.928,-177.965,7.656,148.867
C00591=1139.531,216.947,-64.953,-177.962,7.659,148.867
C00592=1139.527,217.195,-64.979,-177.960,7.661,148.866
C00593=1139.522,217.444,-65.005,-177.957,7.664,148.866
C00594=1139.518,217.693,-65.030,-177.954,7.667,148.866
C00595=1139.513,217.941,-65.055,-177.951,7.669,148.866
C00596=1139.509,218.190,-65.081,-177.948,7.672,148.866
C00597=1139.504,218.438,-65.106,-177.946,7.674,148.866
C00598=1139.500,218.687,-65.132,-177.943,7.677,148.865
C00599=1139.495,218.937,-65.157,-177.940,7.680,148.865
C00600=1139.490,219.185,-65.182,-177.937,7.683,148.865
C00601=1139.486,219.433,-65.208,-177.934,7.686,148.865
C00602=1139.482,219.682,-65.234,-177.931,7.689,148.865
C00603=1139.477,219.930,-65.259,-177.929,7.690,148.865
C00604=1139.473,220.179,-65.285,-177.926,7.693,148.865
C00605=1139.469,220.428,-65.311,-177.923,7.696,148.864
C00606=1139.464,220.676,-65.336,-177.920,7.699,148.864
C00607=1139.459,220.925,-65.361,-177.917,7.702,148.864
C00608=1139.455,221.174,-65.387,-177.914,7.705,148.864
C00609=1139.451,221.423,-65.413,-177.912,7.707,148.864
C00610=1139.446,221.671,-65.438,-177.909,7.710,148.864
C00611=1139.442,221.920,-65.464,-177.906,7.713,148.864
C00612=1139.438,222.169,-65.490,-177.904,7.715,148.864
C00613=1139.432,222.417,-65.516,-177.901,7.718,148.863
C00614=1139.428,222.666,-65.541,-177.897,7.721,148.863
C00615=1139.424,222.915,-65.567,-177.895,7.724,148.863
C00616=1139.419,223.164,-65.593,-177.892,7.726,148.863
C00617=1139.415,223.411,-65.619,-177.890,7.729,148.863
C00618=1139.411,223.660,-65.645,-177.887,7.732,148.863
C00619=1139.406,223.909,-65.670,-177.884,7.735,148.863
C00620=1139.401,224.158,-65.697,-177.881,7.737,148.862
C00621=1139.397,224.406,-65.722,-177.878,7.740,148.862
C00622=1139.392,224.655,-65.748,-177.875,7.743,148.862
C00623=1139.388,224.904,-65.774,-177.872,7.746,148.862
C00624=1139.384,225.152,-65.799,-177.870,7.748,148.862
C00625=1139.379,225.400,-65.826,-177.867,7.751,148.862
C00626=1139.374,225.649,-65.852,-177.865,7.754,148.862
C00627=1139.370,225.898,-65.878,-177.861,7.756,148.861
C00628=1139.366,226.147,-65.903,-177.858,7.759,148.861
C00629=1139.362,226.395,-65.929,-177.856,7.762,148.861
C00630=1139.356,226.643,-65.956,-177.853,7.765,148.861
C00631=1139.352,226.892,-65.982,-177.850,7.768,148.861
C00632=1139.348,227.141,-66.007,-177.848,7.770,148.861
C00633=1139.343,227.390,-66.034,-177.845,7.773,148.861
C00634=1139.339,227.638,-66.060,-177.842,7.776,148.861
C00635=1139.335,227.887,-66.086,-177.839,7.778,148.861
C00636=1139.330,228.135,-66.111,-177.836,7.781,148.860
C00637=1139.325,228.383,-66.138,-177.833,7.784,148.860
C00638=1139.321,228.632,-66.164,-177.831,7.787,148.860
C00639=1139.317,228.881,-66.190,-177.828,7.790,148.860
C00640=1139.312,229.130,-66.217,-177.825,7.793,148.860
C00641=1139.308,229.378,-66.243,-177.822,7.796,148.860
C00642=1139.304,229.627,-66.268,-177.820,7.798,148.860
C00643=1139.299,229.875,-66.295,-177.817,7.801,148.860
C00644=1139.294,230.124,-66.321,-177.814,7.804,148.860
C00645=1139.290,230.372,-66.348,-177.811,7.806,148.859
C00646=1139.286,230.621,-66.374,-177.808,7.809,148.859
C00647=1139.282,230.869,-66.400,-177.805,7.812,148.859
C00648=1139.277,231.118,-66.426,-177.803,7.815,148.859
C00649=1139.273,231.367,-66.453,-177.800,7.818,148.859
C00650=1139.268,231.616,-66.479,-177.797,7.821,148.859
C00651=1139.264,231.864,-66.506,-177.794,7.824,148.859
C00652=1139.259,232.113,-66.532,-177.791,7.827,148.859
C00653=1139.255,232.361,-66.559,-177.789,7.829,148.859
C00654=1139.251,232.610,-66.584,-177.786,7.832,148.859
C00655=1139.246,232.858,-66.611,-177.784,7.835,148.858
C00656=1139.241,233.107,-66.637,-177.781,7.838,148.858
C00657=1139.237,233.355,-66.664,-177.778,7.840,148.858
C00658=1139.233,233.603,-66.690,-177.775,7.843,148.858
C00659=1139.228,233.852,-66.717,-177.772,7.846,148.858
C00660=1139.224,234.101,-66.743,-177.769,7.849,148.858
C00661=1139.219,234.349,-66.770,-177.766,7.852,148.858
C00662=1139.214,234.598,-66.796,-177.764,7.855,148.858
C00663=1139.210,234.846,-66.823,-177.761,7.858,148.858
C00664=1139.206,235.119,-66.853,-177.758,7.861,148.858
C00665=1139.200,235.391,-66.881,-177.755,7.863,148.857
C00666=1139.196,235.662,-66.910,-177.752,7.867,148.857
C00667=1139.191,235.934,-66.940,-177.749,7.870,148.857
C00668=1139.187,236.183,-66.967,-177.746,7.873,148.857
C00669=1139.183,236.432,-66.993,-177.743,7.876,148.857
C00670=1139.178,236.680,-67.020,-177.740,7.879,148.857
C00671=1139.174,236.928,-67.046,-177.737,7.881,148.857
C00672=1139.169,237.177,-67.073,-177.735,7.884,148.857
C00673=1139.164,237.426,-67.099,-177.732,7.887,148.857
C00674=1139.160,237.674,-67.126,-177.729,7.890,148.856
C00675=1139.156,237.923,-67.153,-177.726,7.893,148.856
C00676=1139.151,238.171,-67.180,-177.723,7.896,148.856
C00677=1139.147,238.419,-67.207,-177.721,7.899,148.856
C00678=1139.143,238.668,-67.234,-177.718,7.902,148.856
C00679=1139.138,238.916,-67.261,-177.715,7.905,148.856
C00680=1139.134,239.165,-67.287,-177.712,7.908,148.856
C00681=1139.129,239.413,-67.314,-177.709,7.911,148.856
C00682=1139.124,239.662,-67.341,-177.707,7.913,148.856
C00683=1139.120,239.911,-67.368,-177.704,7.916,148.856
C00684=1139.116,240.160,-67.394,-177.701,7.919,148.856
C00685=1139.112,240.408,-67.421,-177.698,7.922,148.856
C00686=1139.107,240.657,-67.449,-177.696,7.924,148.855
C00687=1139.102,240.905,-67.476,-177.693,7.927,148.855
C00688=1139.098,241.153,-67.502,-177.690,7.930,148.855
C00689=1139.094,241.402,-67.529,-177.688,7.933,148.855
C00690=1139.089,241.650,-67.557,-177.685,7.936,148.855
C00691=1139.085,241.899,-67.584,-177.682,7.939,148.855
C00692=1139.081,242.147,-67.611,-177.679,7.942,148.855
C00693=1139.077,242.395,-67.638,-177.676,7.945,148.855
C00694=1139.072,242.644,-67.665,-177.674,7.948,148.855
C00695=1139.067,242.892,-67.692,-177.671,7.951,148.855
C00696=1139.063,243.141,-67.719,-177.668,7.953,148.855
C00697=1139.059,243.390,-67.746,-177.665,7.956,148.855
C00698=1139.055,243.638,-67.773,-177.662,7.959,148.855
C00699=1139.051,243.886,-67.801,-177.660,7.963,148.855
C00700=1139.046,244.135,-67.828,-177.657,7.965,148.855
C00701=1139.041,244.383,-67.855,-177.654,7.968,148.855
C00702=1139.037,244.632,-67.882,-177.652,7.971,148.854
C00703=1139.032,244.881,-67.909,-177.649,7.974,148.854
C00704=1139.028,245.129,-67.937,-177.646,7.977,148.854
C00705=1139.023,245.377,-67.964,-177.643,7.980,148.854
C00706=1139.019,245.626,-67.992,-177.640,7.983,148.854
C00707=1139.015,245.875,-68.019,-177.637,7.987,148.854
C00708=1139.010,246.123,-68.046,-177.634,7.990,148.854
C00709=1139.006,246.371,-68.073,-177.631,7.992,148.854
C00710=1139.002,246.620,-68.100,-177.629,7.995,148.854
C00711=1138.998,246.868,-68.128,-177.626,7.998,148.854
C00712=1138.993,247.117,-68.155,-177.623,8.001,148.854
C00713=1138.989,247.365,-68.182,-177.620,8.004,148.854
C00714=1138.985,247.614,-68.210,-177.617,8.007,148.854
C00715=1138.980,247.862,-68.237,-177.615,8.010,148.854
C00716=1138.976,248.110,-68.265,-177.612,8.013,148.853
C00717=1138.971,248.359,-68.292,-177.609,8.016,148.854
C00718=1138.967,248.608,-68.320,-177.607,8.019,148.854
C00719=1138.962,248.856,-68.348,-177.604,8.022,148.853
C00720=1138.958,249.104,-68.375,-177.601,8.025,148.853
C00721=1138.954,249.353,-68.403,-177.598,8.028,148.853
C00722=1138.949,249.602,-68.430,-177.595,8.031,148.853
C00723=1138.945,249.849,-68.458,-177.593,8.034,148.853
C00724=1138.941,250.099,-68.486,-177.590,8.037,148.853
C00725=1138.936,250.346,-68.513,-177.587,8.039,148.853
C00726=1138.932,250.595,-68.540,-177.584,8.042,148.853
C00727=1138.928,250.844,-68.569,-177.582,8.045,148.853
C00728=1138.924,251.091,-68.596,-177.579,8.049,148.853
C00729=1138.919,251.340,-68.623,-177.576,8.051,148.853
C00730=1138.914,251.589,-68.652,-177.574,8.054,148.853
C00731=1138.910,251.837,-68.679,-177.571,8.057,148.853
C00732=1138.905,252.085,-68.707,-177.567,8.061,148.853
C00733=1138.902,252.334,-68.735,-177.565,8.064,148.853
C00734=1138.897,252.582,-68.762,-177.562,8.067,148.853
C00735=1138.893,252.831,-68.790,-177.559,8.070,148.853
C00736=1138.888,253.079,-68.819,-177.557,8.073,148.853
C00737=1138.884,253.327,-68.846,-177.554,8.076,148.853
C00738=1138.880,253.576,-68.874,-177.551,8.079,148.853
C00739=1138.875,253.824,-68.902,-177.548,8.082,148.852
C00740=1138.872,254.073,-68.930,-177.545,8.085,148.852
C00741=1138.866,254.321,-68.957,-177.543,8.088,148.852
C00742=1138.863,254.570,-68.986,-177.540,8.091,148.852
C00743=1138.858,254.818,-69.013,-177.537,8.093,148.852
C00744=1138.854,255.066,-69.041,-177.535,8.097,148.852
C00745=1138.849,255.315,-69.069,-177.532,8.100,148.852
C00746=1138.845,255.563,-69.097,-177.529,8.103,148.852
C00747=1138.841,255.812,-69.125,-177.526,8.106,148.852
C00748=1138.836,256.060,-69.153,-177.523,8.109,148.852
C00749=1138.832,256.308,-69.182,-177.520,8.112,148.852
C00750=1138.828,256.556,-69.209,-177.518,8.115,148.852
C00751=1138.823,256.805,-69.238,-177.515,8.118,148.852
C00752=1138.819,257.054,-69.265,-177.512,8.121,148.852
C00753=1138.815,257.302,-69.293,-177.509,8.124,148.852
C00754=1138.810,257.550,-69.322,-177.507,8.127,148.852
C00755=1138.806,257.799,-69.350,-177.504,8.130,148.852
C00756=1138.802,258.047,-69.378,-177.502,8.133,148.852
C00757=1138.797,258.296,-69.406,-177.498,8.137,148.852
C00758=1138.793,258.544,-69.434,-177.495,8.140,148.852
C00759=1138.788,258.792,-69.463,-177.493,8.143,148.852
C00760=1138.784,259.040,-69.491,-177.490,8.146,148.852
C00761=1138.780,259.289,-69.519,-177.487,8.149,148.852
C00762=1138.775,259.537,-69.547,-177.485,8.152,148.852
C00763=1138.771,259.786,-69.575,-177.482,8.155,148.852
C00764=1138.766,260.034,-69.604,-177.479,8.158,148.852
C00765=1138.763,260.282,-69.632,-177.476,8.161,148.852
C00766=1138.758,260.531,-69.661,-177.473,8.165,148.852
C00767=1138.754,260.779,-69.689,-177.471,8.168,148.852
C00768=1138.749,261.052,-69.720,-177.468,8.171,148.852
C00769=1138.745,261.326,-69.751,-177.464,8.174,148.852
C00770=1138.739,261.600,-69.783,-177.462,8.177,148.852
C00771=1138.735,261.873,-69.814,-177.458,8.181,148.852
C00772=1138.730,262.122,-69.843,-177.455,8.184,148.851
C00773=1138.727,262.370,-69.871,-177.453,8.187,148.852
C00774=1138.722,262.618,-69.899,-177.450,8.190,148.852
C00775=1138.718,262.867,-69.927,-177.447,8.193,148.852
C00776=1138.713,263.114,-69.957,-177.445,8.196,148.851
C00777=1138.709,263.363,-69.985,-177.442,8.200,148.852
C00778=1138.705,263.612,-70.013,-177.439,8.203,148.852
C00779=1138.700,263.860,-70.042,-177.436,8.206,148.852
C00780=1138.696,264.108,-70.071,-177.433,8.209,148.851
C00781=1138.692,264.357,-70.099,-177.431,8.212,148.852
C00782=1138.687,264.605,-70.127,-177.428,8.215,148.852
C00783=1138.683,264.853,-70.157,-177.425,8.218,148.851
C00784=1138.679,265.102,-70.185,-177.422,8.222,148.851
C00785=1138.674,265.350,-70.213,-177.420,8.225,148.852
C00786=1138.670,265.598,-70.243,-177.417,8.228,148.852
C00787=1138.666,265.847,-70.271,-177.414,8.231,148.851
C00788=1138.662,266.094,-70.300,-177.411,8.234,148.851
C00789=1138.657,266.343,-70.329,-177.409,8.237,148.852
C00790=1138.653,266.592,-70.357,-177.406,8.240,148.851
C00791=1138.649,266.839,-70.386,-177.403,8.243,148.851
C00792=1138.644,267.088,-70.414,-177.400,8.246,148.851
C00793=1138.640,267.336,-70.444,-177.398,8.250,148.852
C00794=1138.636,267.584,-70.472,-177.395,8.253,148.852
C00795=1138.631,267.833,-70.501,-177.392,8.255,148.851
C00796=1138.627,268.081,-70.530,-177.390,8.259,148.852
C00797=1138.623,268.330,-70.559,-177.386,8.262,148.852
C00798=1138.618,268.578,-70.587,-177.384,8.265,148.852
C00799=1138.614,268.826,-70.617,-177.381,8.268,148.851
C00800=1138.610,269.074,-70.646,-177.378,8.272,148.852
C00801=1138.606,269.323,-70.675,-177.376,8.274,148.852
C00802=1138.601,269.571,-70.704,-177.373,8.277,148.851
C00803=1138.597,269.819,-70.732,-177.370,8.281,148.852
C00804=1138.593,270.067,-70.761,-177.367,8.284,148.852
C00805=1138.589,270.316,-70.791,-177.364,8.287,148.852
C00806=1138.584,270.564,-70.819,-177.362,8.291,148.852
C00807=1138.579,270.812,-70.849,-177.359,8.293,148.852
C00808=1138.576,271.060,-70.878,-177.356,8.297,148.852
C00809=1138.571,271.309,-70.906,-177.353,8.300,148.852
C00810=1138.567,271.557,-70.936,-177.351,8.303,148.852
C00811=1138.563,271.806,-70.965,-177.348,8.306,148.852
C00812=1138.558,272.053,-70.994,-177.346,8.310,148.852
C00813=1138.554,272.302,-71.023,-177.342,8.313,148.852
C00814=1138.550,272.550,-71.053,-177.339,8.316,148.852
C00815=1138.545,272.799,-71.082,-177.337,8.319,148.852
C00816=1138.541,273.047,-71.111,-177.334,8.322,148.852
C00817=1138.538,273.295,-71.140,-177.331,8.325,148.852
C00818=1138.533,273.543,-71.169,-177.329,8.329,148.852
C00819=1138.529,273.791,-71.198,-177.326,8.332,148.852
C00820=1138.524,274.039,-71.228,-177.323,8.335,148.852
C00821=1138.520,274.288,-71.257,-177.321,8.338,148.852
C00822=1138.516,274.536,-71.286,-177.318,8.341,148.852
C00823=1138.512,274.784,-71.316,-177.314,8.345,148.852
C00824=1138.508,275.033,-71.345,-177.312,8.348,148.852
C00825=1138.503,275.281,-71.375,-177.309,8.351,148.852
C00826=1138.499,275.528,-71.404,-177.307,8.355,148.852
C00827=1138.495,275.777,-71.433,-177.304,8.358,148.852
C00828=1138.490,276.025,-71.463,-177.301,8.361,148.852
C00829=1138.486,276.274,-71.492,-177.298,8.364,148.852
C00830=1138.482,276.522,-71.521,-177.296,8.367,148.852
C00831=1138.478,276.770,-71.551,-177.293,8.370,148.852
C00832=1138.474,277.018,-71.581,-177.290,8.374,148.852
C00833=1138.469,277.266,-71.610,-177.287,8.377,148.852
C00834=1138.465,277.515,-71.640,-177.285,8.381,148.853
C00835=1138.460,277.763,-71.670,-177.282,8.384,148.852
C00836=1138.456,278.011,-71.699,-177.279,8.386,148.852
C00837=1138.452,278.260,-71.729,-177.276,8.391,148.853
C00838=1138.448,278.508,-71.758,-177.274,8.393,148.853
C00839=1138.444,278.756,-71.787,-177.271,8.397,148.853
C00840=1138.439,279.004,-71.817,-177.268,8.400,148.853
C00841=1138.435,279.253,-71.846,-177.265,8.404,148.853
C00842=1138.431,279.500,-71.877,-177.263,8.407,148.853
C00843=1138.426,279.749,-71.907,-177.260,8.410,148.853
C00844=1138.422,279.997,-71.936,-177.258,8.413,148.853
C00845=1138.418,280.245,-71.965,-177.254,8.417,148.853
C00846=1138.414,280.494,-71.995,-177.252,8.420,148.853
C00847=1138.410,280.741,-72.025,-177.249,8.423,148.853
C00848=1138.405,280.990,-72.055,-177.247,8.426,148.853
C00849=1138.401,281.238,-72.085,-177.243,8.430,148.853
C00850=1138.397,281.487,-72.114,-177.241,8.433,148.853
C00851=1138.393,281.734,-72.144,-177.238,8.436,148.853
C00852=1138.389,281.982,-72.174,-177.235,8.439,148.853
C00853=1138.384,282.231,-72.204,-177.232,8.443,148.853
C00854=1138.380,282.479,-72.234,-177.230,8.446,148.853
C00855=1138.376,282.727,-72.263,-177.227,8.449,148.854
C00856=1138.371,282.975,-72.293,-177.225,8.452,148.853
C00857=1138.367,283.223,-72.324,-177.222,8.456,148.854
C00858=1138.363,283.471,-72.353,-177.219,8.459,148.854
C00859=1138.359,283.719,-72.383,-177.216,8.462,148.854
C00860=1138.354,283.968,-72.413,-177.213,8.466,148.854
C00861=1138.350,284.215,-72.443,-177.211,8.469,148.854
C00862=1138.346,284.464,-72.473,-177.208,8.472,148.854
C00863=1138.342,284.713,-72.503,-177.206,8.475,148.854
C00864=1138.338,284.960,-72.533,-177.202,8.479,148.854
C00865=1138.333,285.209,-72.563,-177.200,8.482,148.854
C00866=1138.329,285.457,-72.594,-177.197,8.485,148.854
C00867=1138.325,285.705,-72.623,-177.195,8.489,148.854
C00868=1138.320,285.953,-72.654,-177.191,8.492,148.854
C00869=1138.316,286.201,-72.684,-177.189,8.496,148.854
C00870=1138.312,286.449,-72.713,-177.186,8.499,148.854
C00871=1138.308,286.697,-72.745,-177.183,8.503,148.855
C00872=1138.303,286.973,-72.777,-177.181,8.505,148.855
C00873=1138.298,287.249,-72.811,-177.178,8.510,148.855
C00874=1138.294,287.523,-72.845,-177.174,8.513,148.855
C00875=1138.289,287.800,-72.878,-177.171,8.517,148.855
C00876=1138.285,288.047,-72.909,-177.169,8.520,148.855
C00877=1138.281,288.296,-72.940,-177.166,8.524,148.855
C00878=1138.277,288.544,-72.969,-177.163,8.527,148.855
C00879=1138.272,288.792,-73.000,-177.160,8.531,148.855
C00880=1138.268,289.040,-73.030,-177.158,8.533,148.855
C00881=1138.263,289.289,-73.060,-177.155,8.538,148.855
C00882=1138.260,289.537,-73.091,-177.152,8.541,148.856
C00883=1138.255,289.785,-73.121,-177.150,8.544,148.856
C00884=1138.251,290.033,-73.152,-177.147,8.547,148.856
C00885=1138.247,290.281,-73.182,-177.144,8.551,148.856
C00886=1138.243,290.529,-73.212,-177.142,8.554,148.856
C00887=1138.239,290.777,-73.243,-177.139,8.557,148.856
C00888=1138.235,291.025,-73.273,-177.136,8.561,148.856
C00889=1138.230,291.273,-73.304,-177.134,8.564,148.856
C00890=1138.225,291.521,-73.335,-177.131,8.567,148.856
C00891=1138.222,291.769,-73.365,-177.128,8.571,148.856
C00892=1138.218,292.017,-73.396,-177.125,8.574,148.856
C00893=1138.213,292.266,-73.425,-177.123,8.577,148.857
C00894=1138.209,292.514,-73.456,-177.120,8.581,148.857
C00895=1138.205,292.762,-73.487,-177.117,8.584,148.857
C00896=1138.201,293.010,-73.517,-177.115,8.588,148.857
C00897=1138.196,293.258,-73.548,-177.111,8.591,148.857
C00898=1138.192,293.506,-73.579,-177.109,8.595,148.857
C00899=1138.188,293.754,-73.609,-177.107,8.598,148.857
C00900=1138.184,294.002,-73.640,-177.103,8.602,148.857
C00901=1138.180,294.251,-73.671,-177.101,8.605,148.857
C00902=1138.176,294.498,-73.702,-177.098,8.608,148.857
C00903=1138.171,294.746,-73.732,-177.095,8.612,148.858
C00904=1138.167,294.995,-73.763,-177.093,8.615,148.858
C00905=1138.163,295.243,-73.794,-177.090,8.618,148.858
C00906=1138.159,295.490,-73.825,-177.087,8.622,148.858
C00907=1138.155,295.739,-73.856,-177.085,8.625,148.858
C00908=1138.150,295.987,-73.887,-177.081,8.629,148.858
C00909=1138.147,296.235,-73.918,-177.079,8.632,148.858
C00910=1138.143,296.483,-73.948,-177.077,8.636,148.858
C00911=1138.138,296.731,-73.979,-177.073,8.639,148.858
C00912=1138.134,296.980,-74.010,-177.071,8.643,148.859
C00913=1138.130,297.227,-74.042,-177.069,8.646,148.859
C00914=1138.126,297.474,-74.072,-177.065,8.650,148.859
C00915=1138.122,297.723,-74.103,-177.063,8.653,148.859
C00916=1138.117,297.971,-74.134,-177.061,8.656,148.859
C00917=1138.113,298.220,-74.165,-177.057,8.660,148.859
C00918=1138.109,298.467,-74.196,-177.055,8.663,148.859
C00919=1138.104,298.715,-74.227,-177.052,8.667,148.859
C00920=1138.101,298.963,-74.258,-177.050,8.671,148.860
C00921=1138.097,299.211,-74.289,-177.047,8.673,148.860
C00922=1138.093,299.459,-74.320,-177.044,8.678,148.860
C00923=1138.088,299.707,-74.351,-177.041,8.681,148.860
C00924=1138.084,299.955,-74.383,-177.039,8.684,148.860
C00925=1138.080,300.203,-74.414,-177.036,8.688,148.860
C00926=1138.076,300.452,-74.445,-177.033,8.691,148.860
C00927=1138.071,300.699,-74.476,-177.030,8.695,148.861
C00928=1138.067,300.947,-74.507,-177.028,8.698,148.860
C00929=1138.063,301.195,-74.539,-177.025,8.701,148.861
C00930=1138.058,301.443,-74.570,-177.022,8.705,148.861
C00931=1138.055,301.691,-74.601,-177.020,8.708,148.861
C00932=1138.050,301.939,-74.632,-177.017,8.712,148.861
C00933=1138.046,302.188,-74.663,-177.014,8.716,148.861
C00934=1138.042,302.435,-74.695,-177.012,8.719,148.861
C00935=1138.038,302.684,-74.726,-177.009,8.723,148.861
C00936=1138.033,302.931,-74.757,-177.006,8.726,148.862
C00937=1138.030,303.179,-74.789,-177.003,8.730,148.862
C00938=1138.025,303.427,-74.820,-177.001,8.733,148.862
C00939=1138.021,303.675,-74.852,-176.999,8.736,148.862
C00940=1138.017,303.923,-74.883,-176.995,8.740,148.862
C00941=1138.013,304.171,-74.914,-176.993,8.743,148.862
C00942=1138.008,304.419,-74.945,-176.990,8.748,148.863
C00943=1138.005,304.667,-74.977,-176.988,8.751,148.863
C00944=1138.001,304.915,-75.009,-176.985,8.754,148.863
C00945=1137.996,305.163,-75.040,-176.982,8.758,148.863
C00946=1137.993,305.411,-75.072,-176.980,8.761,148.863
C00947=1137.988,305.659,-75.104,-176.977,8.765,148.863
C00948=1137.984,305.908,-75.135,-176.974,8.768,148.863
C00949=1137.979,306.155,-75.166,-176.971,8.772,148.864
C00950=1137.976,306.403,-75.198,-176.969,8.775,148.864
C00951=1137.972,306.651,-75.230,-176.966,8.779,148.864
C00952=1137.967,306.899,-75.261,-176.963,8.783,148.864
C00953=1137.963,307.147,-75.293,-176.961,8.786,148.864
C00954=1137.959,307.395,-75.325,-176.958,8.790,148.864
C00955=1137.955,307.643,-75.356,-176.955,8.793,148.864
C00956=1137.951,307.891,-75.388,-176.952,8.797,148.865
C00957=1137.947,308.139,-75.419,-176.950,8.800,148.865
C00958=1137.942,308.387,-75.452,-176.948,8.803,148.865
C00959=1137.938,308.635,-75.483,-176.945,8.808,148.865
C00960=1137.934,308.883,-75.515,-176.942,8.811,148.865
C00961=1137.930,309.131,-75.547,-176.940,8.815,148.866
C00962=1137.925,309.378,-75.579,-176.937,8.818,148.866
C00963=1137.922,309.626,-75.611,-176.934,8.822,148.866
C00964=1137.918,309.874,-75.642,-176.931,8.825,148.866
C00965=1137.914,310.122,-75.674,-176.929,8.829,148.866
C00966=1137.909,310.371,-75.706,-176.926,8.832,148.866
C00967=1137.905,310.619,-75.737,-176.923,8.837,148.867
C00968=1137.901,310.867,-75.769,-176.921,8.840,148.867
C00969=1137.896,311.114,-75.801,-176.919,8.843,148.867
C00970=1137.893,311.362,-75.833,-176.916,8.847,148.867
C00971=1137.889,311.610,-75.866,-176.913,8.850,148.867
C00972=1137.884,311.857,-75.898,-176.910,8.854,148.867
C00973=1137.881,312.105,-75.930,-176.908,8.857,148.868
C00974=1137.877,312.353,-75.962,-176.905,8.861,148.868
C00975=1137.872,312.602,-75.994,-176.902,8.865,148.868
C00976=1137.868,312.879,-76.030,-176.899,8.869,148.868
C00977=1137.863,313.157,-76.066,-176.896,8.873,148.868
C00978=1137.858,313.435,-76.101,-176.893,8.877,148.869
C00979=1137.854,313.714,-76.137,-176.891,8.881,148.869
C00980=1137.850,313.961,-76.169,-176.888,8.885,148.869
C00981=1137.846,314.209,-76.202,-176.885,8.888,148.869
C00982=1137.842,314.457,-76.234,-176.882,8.892,148.869
C00983=1137.837,314.705,-76.266,-176.880,8.896,148.870
C00984=1137.834,314.953,-76.298,-176.877,8.900,148.870
C00985=1137.829,315.200,-76.331,-176.875,8.903,148.870
C00986=1137.825,315.448,-76.363,-176.871,8.907,148.870
C00987=1137.821,315.697,-76.395,-176.869,8.910,148.870
C00988=1137.817,315.944,-76.428,-176.866,8.914,148.870
C00989=1137.813,316.193,-76.460,-176.864,8.917,148.871
C00990=1137.809,316.440,-76.492,-176.861,8.921,148.871
C00991=1137.805,316.688,-76.525,-176.858,8.925,148.871
C00992=1137.801,316.936,-76.557,-176.856,8.929,148.871
C00993=1137.796,317.184,-76.589,-176.853,8.932,148.871
C00994=1137.793,317.431,-76.622,-176.850,8.936,148.872
C00995=1137.789,317.680,-76.654,-176.848,8.939,148.872
C00996=1137.784,317.927,-76.686,-176.845,8.943,148.872
C00997=1137.780,318.175,-76.719,-176.843,8.947,148.872
C00998=1137.776,318.423,-76.751,-176.840,8.951,148.872
C00999=1137.772,318.671,-76.784,-176.837,8.954,148.873
C01000=1137.768,318.919,-76.816,-176.834,8.958,148.873
C01001=1137.764,319.166,-76.849,-176.833,8.962,148.873
C01002=1137.760,319.415,-76.881,-176.830,8.966,148.874
C01003=1137.757,319.662,-76.914,-176.827,8.969,148.874
C01004=1137.752,319.911,-76.946,-176.824,8.973,148.874
C01005=1137.747,320.158,-76.979,-176.822,8.976,148.874
C01006=1137.744,320.406,-77.011,-176.819,8.980,148.874
C01007=1137.740,320.653,-77.044,-176.816,8.984,148.875
C01008=1137.735,320.901,-77.077,-176.814,8.988,148.875
C01009=1137.732,321.149,-77.109,-176.811,8.992,148.875
C01010=1137.728,321.397,-77.142,-176.808,8.995,148.875
C01011=1137.723,321.645,-77.175,-176.806,8.999,148.875
C01012=1137.720,321.893,-77.207,-176.803,9.002,148.876
C01013=1137.716,322.140,-77.240,-176.800,9.006,148.876
C01014=1137.711,322.389,-77.273,-176.798,9.010,148.876
C01015=1137.707,322.636,-77.306,-176.795,9.014,148.876
C01016=1137.704,322.884,-77.338,-176.793,9.017,148.877
C01017=1137.699,323.132,-77.372,-176.790,9.021,148.877
C01018=1137.695,323.380,-77.404,-176.788,9.025,148.877
C01019=1137.691,323.628,-77.437,-176.785,9.029,148.877
C01020=1137.687,323.875,-77.470,-176.782,9.033,148.877
C01021=1137.683,324.123,-77.503,-176.780,9.036,148.878
C01022=1137.679,324.371,-77.535,-176.777,9.040,148.878
C01023=1137.675,324.619,-77.568,-176.774,9.043,148.878
C01024=1137.671,324.867,-77.602,-176.771,9.047,148.878
C01025=1137.667,325.114,-77.634,-176.769,9.051,148.879
C01026=1137.663,325.362,-77.667,-176.767,9.055,148.879
C01027=1137.659,325.609,-77.700,-176.764,9.059,148.879
C01028=1137.655,325.857,-77.734,-176.761,9.062,148.879
C01029=1137.650,326.106,-77.766,-176.758,9.066,148.880
C01030=1137.646,326.353,-77.799,-176.756,9.070,148.880
C01031=1137.642,326.601,-77.832,-176.753,9.074,148.880
C01032=1137.638,326.849,-77.866,-176.751,9.077,148.880
C01033=1137.635,327.096,-77.898,-176.748,9.081,148.881
C01034=1137.630,327.344,-77.931,-176.745,9.085,148.881
C01035=1137.626,327.592,-77.964,-176.743,9.089,148.881
C01036=1137.622,327.839,-77.998,-176.740,9.093,148.881
C01037=1137.619,328.088,-78.031,-176.738,9.096,148.882
C01038=1137.614,328.336,-78.064,-176.735,9.100,148.882
C01039=1137.610,328.583,-78.097,-176.733,9.104,148.882
C01040=1137.606,328.831,-78.131,-176.730,9.108,148.882
C01041=1137.602,329.079,-78.164,-176.727,9.112,148.883
C01042=1137.598,329.326,-78.197,-176.725,9.115,148.883
C01043=1137.594,329.574,-78.231,-176.722,9.119,148.883
C01044=1137.590,329.821,-78.264,-176.720,9.123,148.883
C01045=1137.586,330.069,-78.297,-176.717,9.127,148.884
C01046=1137.582,330.317,-78.331,-176.714,9.131,148.884
C01047=1137.578,330.565,-78.364,-176.712,9.134,148.884
C01048=1137.574,330.813,-78.397,-176.709,9.138,148.884
C01049=1137.570,331.060,-78.431,-176.707,9.142,148.885
C01050=1137.566,331.308,-78.464,-176.704,9.146,148.885
C01051=1137.562,331.555,-78.497,-176.701,9.150,148.885
C01052=1137.557,331.803,-78.531,-176.699,9.153,148.886
C01053=1137.554,332.051,-78.565,-176.696,9.157,148.886
C01054=1137.550,332.299,-78.598,-176.693,9.162,148.886
C01055=1137.545,332.547,-78.631,-176.691,9.165,148.886
C01056=1137.541,332.794,-78.665,-176.688,9.169,148.887
C01057=1137.537,333.042,-78.698,-176.686,9.172,148.887
C01058=1137.534,333.290,-78.732,-176.683,9.177,148.887
C01059=1137.530,333.538,-78.765,-176.680,9.181,148.888
C01060=1137.525,333.785,-78.800,-176.678,9.184,148.888
C01061=1137.521,334.033,-78.833,-176.676,9.189,148.888
C01062=1137.517,334.280,-78.867,-176.673,9.193,148.888
C01063=1137.514,334.528,-78.900,-176.670,9.196,148.889
C01064=1137.510,334.776,-78.933,-176.668,9.200,148.889
C01065=1137.506,335.023,-78.967,-176.665,9.204,148.889
C01066=1137.501,335.271,-79.001,-176.662,9.208,148.889
C01067=1137.498,335.519,-79.035,-176.660,9.212,148.890
C01068=1137.494,335.767,-79.068,-176.658,9.215,148.890
C01069=1137.490,336.014,-79.102,-176.655,9.219,148.890
C01070=1137.485,336.262,-79.136,-176.652,9.224,148.891
C01071=1137.482,336.510,-79.170,-176.650,9.227,148.891
C01072=1137.477,336.758,-79.203,-176.647,9.231,148.891
C01073=1137.474,337.005,-79.237,-176.644,9.235,148.892
C01074=1137.469,337.253,-79.271,-176.642,9.239,148.892
C01075=1137.465,337.501,-79.305,-176.639,9.243,148.892
C01076=1137.462,337.748,-79.339,-176.637,9.247,148.893
C01077=1137.457,337.996,-79.373,-176.634,9.250,148.893
C01078=1137.454,338.243,-79.407,-176.631,9.254,148.893
C01079=1137.450,338.491,-79.441,-176.629,9.258,148.893
C01080=1137.445,338.772,-79.479,-176.626,9.263,148.894
C01081=1137.441,339.053,-79.518,-176.623,9.267,148.894
C01082=1137.436,339.334,-79.556,-176.620,9.271,148.894
C01083=1137.431,339.614,-79.594,-176.617,9.277,148.895
C01084=1137.428,339.862,-79.629,-176.615,9.280,148.895
C01085=1137.423,340.110,-79.663,-176.612,9.284,148.895
C01086=1137.419,340.357,-79.697,-176.610,9.288,148.896
C01087=1137.415,340.605,-79.731,-176.607,9.291,148.896
C01088=1137.411,340.853,-79.765,-176.605,9.296,148.896
C01089=1137.407,341.100,-79.800,-176.602,9.300,148.897
C01090=1137.404,341.348,-79.834,-176.600,9.304,148.897
C01091=1137.399,341.595,-79.868,-176.597,9.308,148.897
C01092=1137.395,341.842,-79.902,-176.594,9.312,148.898
C01093=1137.392,342.091,-79.936,-176.592,9.315,148.898
C01094=1137.387,342.338,-79.970,-176.589,9.319,148.898
C01095=1137.384,342.586,-80.004,-176.587,9.324,148.899
C01096=1137.379,342.833,-80.039,-176.584,9.328,148.899
C01097=1137.375,343.080,-80.073,-176.582,9.331,148.899
C01098=1137.371,343.329,-80.107,-176.579,9.335,148.899
C01099=1137.367,343.576,-80.142,-176.576,9.340,148.900
C01100=1137.364,343.824,-80.176,-176.574,9.343,148.900
C01101=1137.359,344.071,-80.211,-176.571,9.347,148.901
C01102=1137.356,344.319,-80.245,-176.568,9.351,148.901
C01103=1137.351,344.566,-80.279,-176.567,9.355,148.901
C01104=1137.348,344.814,-80.314,-176.564,9.359,148.901
C01105=1137.343,345.062,-80.348,-176.561,9.363,148.902
C01106=1137.339,345.309,-80.383,-176.558,9.368,148.902
C01107=1137.336,345.557,-80.417,-176.556,9.371,148.903
C01108=1137.331,345.804,-80.451,-176.553,9.375,148.903
C01109=1137.328,346.052,-80.485,-176.551,9.380,148.903
C01110=1137.323,346.300,-80.520,-176.548,9.383,148.903
C01111=1137.320,346.547,-80.555,-176.546,9.387,148.904
C01112=1137.316,346.794,-80.589,-176.543,9.391,148.904
C01113=1137.312,347.042,-80.624,-176.540,9.396,148.905
C01114=1137.307,347.290,-80.659,-176.539,9.399,148.905
C01115=1137.304,347.538,-80.693,-176.536,9.403,148.905
C01116=1137.300,347.786,-80.728,-176.533,9.408,148.906
C01117=1137.296,348.032,-80.763,-176.531,9.411,148.906
C01118=1137.293,348.280,-80.797,-176.528,9.415,148.906
C01119=1137.288,348.528,-80.832,-176.525,9.419,148.907
C01120=1137.282,348.897,-80.884,-176.522,9.425,148.907
C01121=1137.261,350.252,-81.075,-177.295,10.940,149.500
C01122=1137.257,350.499,-81.110,-177.291,10.942,149.500
C01123=1137.253,350.747,-81.145,-177.287,10.946,149.500
C01124=1137.249,350.994,-81.180,-177.283,10.949,149.499
C01125=1137.245,351.242,-81.216,-177.280,10.951,149.499
C01126=1137.241,351.489,-81.250,-177.276,10.954,149.499
C01127=1137.237,351.736,-81.286,-177.272,10.956,149.499
C01128=1137.233,351.984,-81.322,-177.269,10.959,149.498
C01129=1137.230,352.232,-81.356,-177.265,10.962,149.498
C01130=1137.225,352.479,-81.392,-177.261,10.964,149.498
C01131=1137.222,352.726,-81.427,-177.257,10.967,149.498
C01132=1137.218,352.974,-81.463,-177.254,10.970,149.497
C01133=1137.213,353.221,-81.497,-177.250,10.973,149.497
C01134=1137.210,353.469,-81.533,-177.246,10.975,149.497
C01135=1137.206,353.716,-81.568,-177.243,10.978,149.497
C01136=1137.202,353.964,-81.604,-177.239,10.981,149.496
C01137=1137.199,354.211,-81.639,-177.235,10.983,149.496
C01138=1137.194,354.458,-81.675,-177.232,10.986,149.496
C01139=1137.191,354.706,-81.710,-177.228,10.988,149.495
C01140=1137.186,354.954,-81.745,-177.224,10.991,149.495
C01141=1137.182,355.202,-81.781,-177.221,10.993,149.495
C01142=1137.179,355.449,-81.817,-177.217,10.996,149.495
C01143=1137.174,355.696,-81.852,-177.213,10.999,149.494
C01144=1137.171,355.943,-81.887,-177.210,11.001,149.494
C01145=1137.167,356.191,-81.923,-177.206,11.004,149.494
C01146=1137.164,356.438,-81.958,-177.202,11.007,149.494
C01147=1137.160,356.686,-81.994,-177.199,11.009,149.493
C01148=1137.155,356.934,-82.030,-177.195,11.011,149.493
C01149=1137.151,357.180,-82.065,-177.192,11.014,149.493
C01150=1137.148,357.428,-82.101,-177.188,11.017,149.492
C01151=1137.144,357.675,-82.137,-177.184,11.019,149.492
C01152=1137.141,357.922,-82.173,-177.181,11.022,149.492
C01153=1137.136,358.170,-82.209,-177.178,11.024,149.492
C01154=1137.132,358.418,-82.244,-177.174,11.026,149.491
C01155=1137.129,358.665,-82.280,-177.171,11.029,149.491
C01156=1137.125,358.913,-82.315,-177.167,11.032,149.491
C01157=1137.120,359.160,-82.351,-177.163,11.034,149.490
C01158=1137.117,359.407,-82.387,-177.160,11.036,149.490
C01159=1137.113,359.654,-82.423,-177.157,11.039,149.490
C01160=1137.109,359.902,-82.459,-177.153,11.041,149.490
C01161=1137.105,360.149,-82.495,-177.150,11.044,149.489
C01162=1137.102,360.396,-82.531,-177.146,11.046,149.489
C01163=1137.098,360.644,-82.567,-177.143,11.048,149.489
C01164=1137.094,360.892,-82.603,-177.140,11.051,149.489
C01165=1137.090,361.139,-82.638,-177.136,11.053,149.488
C01166=1137.087,361.386,-82.674,-177.133,11.056,149.488
C01167=1137.083,361.633,-82.710,-177.129,11.058,149.488
C01168=1137.079,361.881,-82.746,-177.126,11.060,149.488
C01169=1137.074,362.172,-82.788,-177.122,11.063,149.487
C01170=1137.070,362.463,-82.831,-177.117,11.066,149.487
C01171=1137.065,362.755,-82.874,-177.114,11.069,149.487
C01172=1137.061,363.046,-82.916,-177.110,11.072,149.486
C01173=1137.056,363.294,-82.952,-177.106,11.074,149.486
C01174=1137.053,363.541,-82.988,-177.103,11.077,149.486
C01175=1137.049,363.789,-83.025,-177.100,11.079,149.486
C01176=1137.045,364.036,-83.061,-177.097,11.082,149.486
C01177=1137.042,364.283,-83.096,-177.093,11.083,149.485
C01178=1137.038,364.531,-83.133,-177.090,11.085,149.485
C01179=1137.034,364.778,-83.169,-177.087,11.088,149.485
C01180=1137.030,365.025,-83.206,-177.084,11.090,149.484
C01181=1137.026,365.273,-83.241,-177.080,11.093,149.484
C01182=1137.022,365.520,-83.278,-177.077,11.095,149.484
C01183=1137.018,365.767,-83.314,-177.074,11.098,149.484
C01184=1137.014,366.015,-83.350,-177.071,11.099,149.484
C01185=1137.012,366.262,-83.387,-177.068,11.102,149.483
C01186=1137.007,366.510,-83.423,-177.064,11.104,149.483
C01187=1137.004,366.757,-83.460,-177.061,11.107,149.483
C01188=1136.999,367.005,-83.496,-177.057,11.109,149.482
C01189=1136.996,367.252,-83.532,-177.055,11.111,149.482
C01190=1136.992,367.499,-83.569,-177.051,11.113,149.482
C01191=1136.988,367.746,-83.604,-177.048,11.116,149.482
C01192=1136.984,367.993,-83.641,-177.045,11.118,149.482
C01193=1136.980,368.241,-83.678,-177.042,11.120,149.481
C01194=1136.977,368.487,-83.714,-177.039,11.122,149.481
C01195=1136.972,368.735,-83.750,-177.036,11.125,149.481
C01196=1136.969,368.982,-83.787,-177.033,11.128,149.481
C01197=1136.965,369.230,-83.824,-177.030,11.129,149.481
C01198=1136.961,369.477,-83.861,-177.027,11.132,149.480
C01199=1136.958,369.725,-83.896,-177.023,11.134,149.480
C01200=1136.954,369.972,-83.933,-177.021,11.136,149.480
C01201=1136.950,370.219,-83.970,-177.017,11.138,149.480
C01202=1136.946,370.466,-84.006,-177.014,11.141,149.480
C01203=1136.942,370.713,-84.043,-177.011,11.143,149.479
C01204=1136.938,370.960,-84.080,-177.008,11.145,149.479
C01205=1136.935,371.208,-84.117,-177.006,11.147,149.479
C01206=1136.931,371.456,-84.153,-177.003,11.150,149.479
C01207=1136.927,371.703,-84.190,-176.999,11.152,149.479
C01208=1136.923,371.950,-84.226,-176.997,11.154,149.478
C01209=1136.919,372.197,-84.263,-176.993,11.156,149.478
C01210=1136.915,372.444,-84.300,-176.991,11.158,149.478
C01211=1136.912,372.692,-84.336,-176.988,11.161,149.478
C01212=1136.908,372.939,-84.373,-176.984,11.163,149.478
C01213=1136.904,373.186,-84.410,-176.982,11.165,149.477
C01214=1136.900,373.433,-84.447,-176.979,11.168,149.477
C01215=1136.897,373.680,-84.483,-176.976,11.169,149.477
C01216=1136.893,373.928,-84.520,-176.973,11.172,149.477
C01217=1136.889,374.175,-84.557,-176.971,11.174,149.477
C01218=1136.885,374.423,-84.594,-176.967,11.176,149.477
C01219=1136.881,374.670,-84.631,-176.965,11.178,149.476
C01220=1136.878,374.917,-84.667,-176.962,11.181,149.476
C01221=1136.874,375.130,-84.699,-176.959,11.183,149.476
C01222=1136.871,375.343,-84.731,-176.957,11.185,149.476
C01223=1136.868,375.555,-84.763,-176.954,11.187,149.476
C01224=1136.865,375.769,-84.796,-176.952,11.188,149.476
C01225=1136.862,375.982,-84.827,-176.950,11.190,149.476
C01226=1136.858,376.195,-84.859,-176.947,11.192,149.476
C01227=1136.856,376.408,-84.890,-176.945,11.194,149.476
C01228=1136.852,376.621,-84.922,-176.942,11.196,149.475
C01229=1136.848,376.868,-84.959,-176.940,11.198,149.475
C01230=1136.844,377.115,-84.997,-176.937,11.201,149.475
C01231=1136.840,377.363,-85.034,-176.934,11.203,149.475
C01232=1136.836,377.610,-85.071,-176.932,11.205,149.475
C01233=1136.833,377.857,-85.107,-176.929,11.207,149.475
C01234=1136.829,378.105,-85.144,-176.927,11.209,149.475
C01235=1136.826,378.351,-85.182,-176.923,11.212,149.475
C01236=1136.822,378.598,-85.219,-176.921,11.214,149.475
C01237=1136.818,378.846,-85.256,-176.919,11.216,149.474
C01238=1136.814,379.093,-85.293,-176.915,11.218,149.474
C01239=1136.810,379.340,-85.330,-176.913,11.220,149.474
C01240=1136.806,379.587,-85.367,-176.911,11.222,149.474
C01241=1136.803,379.835,-85.404,-176.908,11.225,149.474
C01242=1136.799,380.082,-85.442,-176.905,11.227,149.474
C01243=1136.795,380.329,-85.479,-176.903,11.229,149.474
C01244=1136.791,380.577,-85.516,-176.900,11.232,149.474
C01245=1136.787,380.823,-85.554,-176.898,11.234,149.474
C01246=1136.783,381.070,-85.590,-176.896,11.236,149.474
C01247=1136.780,381.318,-85.628,-176.893,11.238,149.474
C01248=1136.776,381.565,-85.665,-176.890,11.240,149.474
C01249=1136.772,381.812,-85.702,-176.888,11.242,149.474
C01250=1136.769,382.059,-85.740,-176.885,11.245,149.474
C01251=1136.765,382.307,-85.777,-176.883,11.247,149.474
C01252=1136.761,382.554,-85.815,-176.881,11.249,149.473
C01253=1136.757,382.801,-85.852,-176.878,11.251,149.473
C01254=1136.754,383.048,-85.889,-176.876,11.254,149.473
C01255=1136.750,383.296,-85.927,-176.873,11.256,149.473
C01256=1136.746,383.542,-85.964,-176.872,11.257,149.473
C01257=1136.742,383.789,-86.001,-176.871,11.259,149.474
C01258=1136.739,384.037,-86.039,-176.870,11.261,149.474
C01259=1136.735,384.284,-86.076,-176.869,11.262,149.474
C01260=1136.732,384.531,-86.114,-176.868,11.264,149.474
C01261=1136.728,384.778,-86.151,-176.867,11.264,149.474
C01262=1136.724,385.025,-86.188,-176.867,11.266,149.474
C01263=1136.720,385.273,-86.225,-176.866,11.268,149.475
C01264=1136.717,385.519,-86.263,-176.865,11.269,149.475
C01265=1136.713,385.767,-86.300,-176.864,11.271,149.475
C01266=1136.709,386.014,-86.338,-176.864,11.272,149.475
C01267=1136.705,386.261,-86.376,-176.863,11.274,149.475
C01268=1136.701,386.508,-86.413,-176.862,11.275,149.475
C01269=1136.697,386.755,-86.451,-176.862,11.277,149.476
C01270=1136.694,387.003,-86.488,-176.861,11.279,149.476
C01271=1136.690,387.249,-86.525,-176.861,11.280,149.476
C01272=1136.686,387.497,-86.562,-176.860,11.282,149.476
C01273=1136.683,387.744,-86.600,-176.859,11.283,149.477
C01274=1136.679,387.991,-86.638,-176.859,11.285,149.477
C01275=1136.676,388.238,-86.675,-176.858,11.286,149.477
C01276=1136.672,388.485,-86.713,-176.858,11.288,149.477
C01277=1136.668,388.698,-86.745,-176.857,11.289,149.478
C01278=1136.665,388.911,-86.777,-176.857,11.291,149.478
C01279=1136.661,389.124,-86.809,-176.857,11.292,149.478
C01280=1136.659,389.337,-86.842,-176.856,11.294,149.479
C01281=1136.655,389.549,-86.875,-176.856,11.295,149.479
C01282=1136.653,389.763,-86.907,-176.855,11.297,149.479
C01283=1136.649,389.975,-86.939,-176.855,11.298,149.480
C01284=1136.646,390.189,-86.971,-176.855,11.300,149.480
C01285=1136.642,390.435,-87.009,-176.854,11.302,149.480
C01286=1136.639,390.683,-87.047,-176.854,11.303,149.480
C01287=1136.635,390.930,-87.084,-176.854,11.305,149.481
C01288=1136.630,391.177,-87.122,-176.853,11.307,149.481
C01289=1136.627,391.425,-87.159,-176.853,11.308,149.482
C01290=1136.623,391.671,-87.197,-176.852,11.311,149.482
C01291=1136.620,391.918,-87.235,-176.853,11.312,149.483
C01292=1136.616,392.166,-87.271,-176.852,11.314,149.483
C01293=1136.613,392.413,-87.309,-176.852,11.317,149.483
C01294=1136.609,392.659,-87.347,-176.852,11.318,149.484
C01295=1136.605,392.907,-87.386,-176.851,11.320,149.484
C01296=1136.601,393.154,-87.422,-176.851,11.322,149.485
C01297=1136.597,393.401,-87.460,-176.851,11.324,149.485
C01298=1136.594,393.648,-87.498,-176.852,11.326,149.486
C01299=1136.590,393.895,-87.535,-176.851,11.328,149.486
C01300=1136.587,394.142,-87.573,-176.851,11.330,149.487
C01301=1136.582,394.389,-87.611,-176.851,11.332,149.487
C01302=1136.578,394.637,-87.648,-176.851,11.334,149.488
C01303=1136.575,394.884,-87.686,-176.851,11.336,149.488
C01304=1136.572,395.131,-87.724,-176.851,11.338,149.489
C01305=1136.567,395.378,-87.760,-176.851,11.341,149.489
C01306=1136.563,395.625,-87.799,-176.851,11.342,149.490
C01307=1136.560,395.872,-87.837,-176.851,11.345,149.491
C01308=1136.556,396.119,-87.874,-176.852,11.347,149.491
C01309=1136.552,396.367,-87.911,-176.852,11.349,149.492
C01310=1136.549,396.613,-87.949,-176.852,11.352,149.493
C01311=1136.545,396.861,-87.987,-176.852,11.354,149.493
C01312=1136.541,397.108,-88.025,-176.852,11.356,149.494
C01313=1136.537,397.356,-88.062,-176.853,11.358,149.494
C01314=1136.534,397.602,-88.100,-176.853,11.361,149.495
C01315=1136.530,397.849,-88.138,-176.853,11.363,149.496
C01316=1136.526,398.096,-88.176,-176.853,11.365,149.496
C01317=1136.522,398.344,-88.213,-176.853,11.368,149.497
C01318=1136.519,398.591,-88.251,-176.854,11.370,149.498
C01319=1136.515,398.837,-88.288,-176.854,11.372,149.499
C01320=1136.512,399.085,-88.326,-176.854,11.375,149.499
C01321=1136.507,399.332,-88.364,-176.855,11.377,149.500
C01322=1136.504,399.579,-88.402,-176.855,11.380,149.501
C01323=1136.500,399.826,-88.439,-176.855,11.383,149.502
C01324=1136.497,400.073,-88.477,-176.856,11.385,149.502
C01325=1136.493,400.320,-88.515,-176.857,11.388,149.503
C01326=1136.489,400.568,-88.553,-176.858,11.390,149.504
C01327=1136.485,400.815,-88.590,-176.858,11.393,149.505
C01328=1136.482,401.062,-88.628,-176.858,11.395,149.506
C01329=1136.478,401.308,-88.666,-176.859,11.398,149.506
C01330=1136.474,401.557,-88.703,-176.860,11.400,149.507
C01331=1136.470,401.803,-88.741,-176.860,11.403,149.508
C01332=1136.467,402.050,-88.779,-176.861,11.406,149.509
C01333=1136.463,402.263,-88.812,-176.861,11.408,149.510
C01334=1136.460,402.476,-88.845,-176.862,11.410,149.510
C01335=1136.457,402.689,-88.876,-176.862,11.413,149.511
C01336=1136.454,402.902,-88.909,-176.863,11.415,149.512
C01337=1136.450,403.114,-88.942,-176.864,11.418,149.513
C01338=1136.447,403.328,-88.974,-176.865,11.420,149.514
C01339=1136.444,403.540,-89.006,-176.866,11.423,149.514
C01340=1136.441,403.752,-89.039,-176.866,11.425,149.515
C01341=1136.437,404.000,-89.077,-176.867,11.429,149.516
C01342=1136.433,404.246,-89.115,-176.868,11.431,149.517
C01343=1136.430,404.494,-89.152,-176.868,11.434,149.518
C01344=1136.426,404.741,-89.190,-176.869,11.437,149.519
C01345=1136.422,404.988,-89.228,-176.870,11.440,149.520
C01346=1136.418,405.235,-89.266,-176.871,11.443,149.521
C01347=1136.415,405.482,-89.304,-176.872,11.446,149.522
C01348=1136.411,405.729,-89.341,-176.874,11.449,149.523
C01349=1136.407,405.977,-89.379,-176.874,11.452,149.524
C01350=1136.403,406.224,-89.417,-176.875,11.456,149.526
C01351=1136.400,406.471,-89.455,-176.876,11.459,149.527
C01352=1136.396,406.717,-89.492,-176.878,11.462,149.528
C01353=1136.392,406.965,-89.531,-176.878,11.465,149.529
C01354=1136.388,407.212,-89.568,-176.880,11.468,149.530
C01355=1136.385,407.459,-89.606,-176.881,11.471,149.531
C01356=1136.382,407.707,-89.643,-176.882,11.475,149.532
C01357=1136.377,407.954,-89.682,-176.883,11.478,149.533
C01358=1136.374,408.201,-89.720,-176.885,11.482,149.535
C01359=1136.370,408.447,-89.757,-176.886,11.484,149.536
C01360=1136.367,408.695,-89.795,-176.887,11.488,149.537
C01361=1136.363,408.942,-89.833,-176.888,11.492,149.538
C01362=1136.359,409.189,-89.871,-176.890,11.495,149.539
C01363=1136.356,409.435,-89.909,-176.891,11.499,149.541
C01364=1136.351,409.684,-89.947,-176.893,11.502,149.542
C01365=1136.348,409.930,-89.984,-176.894,11.505,149.543
C01366=1136.344,410.178,-90.022,-176.895,11.509,149.544
C01367=1136.341,410.424,-90.060,-176.897,11.513,149.546
C01368=1136.337,410.672,-90.098,-176.898,11.517,149.547
C01369=1136.333,410.918,-90.136,-176.900,11.520,149.548
C01370=1136.330,411.165,-90.174,-176.902,11.524,149.550
C01371=1136.325,411.412,-90.212,-176.903,11.527,149.551
C01372=1136.322,411.660,-90.249,-176.904,11.531,149.553
C01373=1136.318,411.907,-90.287,-176.906,11.535,149.554
C01374=1136.315,412.154,-90.325,-176.908,11.538,149.555
C01375=1136.310,412.401,-90.363,-176.910,11.542,149.557
C01376=1136.307,412.648,-90.401,-176.911,11.546,149.558
C01377=1136.303,412.895,-90.438,-176.913,11.550,149.560
C01378=1136.299,413.142,-90.477,-176.914,11.554,149.561
C01379=1136.295,413.389,-90.514,-176.916,11.558,149.563
C01380=1136.292,413.636,-90.552,-176.918,11.562,149.564
C01381=1136.288,413.883,-90.589,-176.920,11.567,149.565
C01382=1136.284,414.131,-90.628,-176.922,11.570,149.567
C01383=1136.280,414.378,-90.665,-176.924,11.574,149.569
C01384=1136.277,414.625,-90.703,-176.926,11.578,149.570
C01385=1136.276,414.872,-90.742,-176.928,11.583,149.572
C01386=1136.273,415.119,-90.779,-176.930,11.587,149.573
C01387=1136.272,415.366,-90.816,-176.931,11.591,149.575
C01388=1136.273,415.613,-90.854,-176.933,11.595,149.576
C01389=1136.272,415.826,-90.886,-176.935,11.598,149.578
C01390=1136.273,416.038,-90.918,-176.937,11.603,149.579
C01391=1136.274,416.251,-90.950,-176.939,11.606,149.581
C01392=1136.275,416.464,-90.981,-176.941,11.610,149.582
C01393=1136.277,416.677,-91.013,-176.943,11.614,149.584
C01394=1136.279,416.890,-91.045,-176.945,11.617,149.585
C01395=1136.282,417.103,-91.077,-176.947,11.621,149.586
C01396=1136.286,417.315,-91.109,-176.949,11.624,149.588
C01397=1135.867,417.314,-91.171,-176.941,11.630,149.587
C01398=1135.863,417.102,-91.140,-176.939,11.625,149.586
C01399=1135.861,416.890,-91.108,-176.937,11.621,149.584
C01400=1135.858,416.677,-91.076,-176.935,11.618,149.583
C01401=1135.856,416.464,-91.044,-176.934,11.614,149.581
C01402=1135.855,416.251,-91.013,-176.931,11.611,149.580
C01403=1135.854,416.038,-90.980,-176.930,11.607,149.579
C01404=1135.853,415.826,-90.949,-176.928,11.603,149.577
C01405=1135.852,415.613,-90.917,-176.926,11.600,149.576
C01406=1135.853,415.366,-90.879,-176.924,11.595,149.574
C01407=1135.854,415.119,-90.842,-176.922,11.591,149.572
C01408=1135.856,414.872,-90.803,-176.920,11.587,149.571
C01409=1135.858,414.625,-90.766,-176.918,11.583,149.569
C01410=1135.861,414.378,-90.728,-176.917,11.578,149.568
C01411=1135.865,414.130,-90.690,-176.915,11.575,149.566
C01412=1135.868,413.884,-90.653,-176.913,11.570,149.565
C01413=1135.872,413.636,-90.614,-176.911,11.566,149.563
C01414=1135.876,413.390,-90.576,-176.910,11.562,149.562
C01415=1135.879,413.142,-90.538,-176.908,11.558,149.560
C01416=1135.884,412.895,-90.500,-176.907,11.554,149.559
C01417=1135.887,412.648,-90.462,-176.905,11.550,149.557
C01418=1135.891,412.401,-90.426,-176.903,11.546,149.556
C01419=1135.895,412.153,-90.387,-176.902,11.542,149.555
C01420=1135.899,411.907,-90.349,-176.900,11.538,149.553
C01421=1135.902,411.660,-90.311,-176.898,11.535,149.552
C01422=1135.906,411.413,-90.274,-176.897,11.531,149.551
C01423=1135.910,411.165,-90.235,-176.895,11.527,149.549
C01424=1135.913,410.918,-90.197,-176.894,11.524,149.548
C01425=1135.917,410.672,-90.160,-176.893,11.520,149.547
C01426=1135.921,410.424,-90.121,-176.891,11.516,149.545
C01427=1135.924,410.177,-90.084,-176.890,11.512,149.544
C01428=1135.928,409.930,-90.046,-176.889,11.509,149.543
C01429=1135.932,409.683,-90.008,-176.886,11.506,149.541
C01430=1135.936,409.435,-89.970,-176.885,11.502,149.540
C01431=1135.939,409.189,-89.933,-176.884,11.499,149.539
C01432=1135.943,408.942,-89.895,-176.883,11.495,149.538
C01433=1135.947,408.695,-89.857,-176.882,11.491,149.536
C01434=1135.950,408.447,-89.819,-176.881,11.488,149.535
C01435=1135.954,408.201,-89.781,-176.879,11.485,149.534
C01436=1135.958,407.953,-89.743,-176.878,11.481,149.533
C01437=1135.962,407.707,-89.705,-176.877,11.478,149.532
C01438=1135.965,407.459,-89.668,-176.876,11.474,149.531
C01439=1135.969,407.212,-89.630,-176.875,11.471,149.529
C01440=1135.973,406.965,-89.592,-176.873,11.468,149.528
C01441=1135.977,406.718,-89.554,-176.872,11.465,149.527
C01442=1135.980,406.471,-89.516,-176.871,11.461,149.526
C01443=1135.984,406.224,-89.479,-176.871,11.458,149.525
C01444=1135.988,405.977,-89.440,-176.870,11.455,149.524
C01445=1135.992,405.730,-89.403,-176.868,11.452,149.523
C01446=1135.995,405.482,-89.365,-176.867,11.449,149.522
C01447=1135.999,405.236,-89.328,-176.867,11.446,149.521
C01448=1136.003,404.988,-89.289,-176.866,11.443,149.520
C01449=1136.007,404.741,-89.252,-176.865,11.440,149.519
C01450=1136.010,404.494,-89.214,-176.864,11.437,149.518
C01451=1136.014,404.247,-89.176,-176.863,11.434,149.517
C01452=1136.017,404.000,-89.138,-176.863,11.430,149.516
C01453=1136.022,403.753,-89.101,-176.861,11.428,149.515
C01454=1136.024,403.540,-89.068,-176.861,11.425,149.514
C01455=1136.028,403.327,-89.035,-176.860,11.423,149.513
C01456=1136.031,403.114,-89.002,-176.860,11.420,149.512
C01457=1136.035,402.901,-88.970,-176.859,11.418,149.512
C01458=1136.037,402.688,-88.937,-176.859,11.415,149.511
C01459=1136.041,402.476,-88.905,-176.858,11.413,149.510
C01460=1136.043,402.263,-88.873,-176.858,11.410,149.509
C01461=1136.047,402.050,-88.841,-176.857,11.408,149.509
C01462=1136.051,401.803,-88.802,-176.856,11.405,149.508
C01463=1136.055,401.556,-88.765,-176.856,11.403,149.507
C01464=1136.058,401.309,-88.727,-176.855,11.400,149.506
C01465=1136.062,401.062,-88.689,-176.855,11.398,149.505
C01466=1136.065,400.815,-88.650,-176.854,11.395,149.504
C01467=1136.070,400.568,-88.614,-176.853,11.393,149.504
C01468=1136.073,400.320,-88.576,-176.853,11.390,149.503
C01469=1136.077,400.074,-88.538,-176.853,11.387,149.502
C01470=1136.080,399.826,-88.500,-176.852,11.385,149.501
C01471=1136.084,399.580,-88.462,-176.852,11.382,149.501
C01472=1136.088,399.332,-88.425,-176.852,11.379,149.500
C01473=1136.092,399.085,-88.387,-176.851,11.377,149.499
C01474=1136.095,398.839,-88.350,-176.851,11.375,149.498
C01475=1136.099,398.591,-88.311,-176.851,11.372,149.498
C01476=1136.103,398.344,-88.274,-176.850,11.370,149.497
C01477=1136.107,398.096,-88.236,-176.850,11.367,149.496
C01478=1136.110,397.850,-88.199,-176.850,11.365,149.496
C01479=1136.113,397.603,-88.161,-176.849,11.363,149.495
C01480=1136.118,397.356,-88.123,-176.849,11.360,149.494
C01481=1136.122,397.108,-88.085,-176.849,11.358,149.493
C01482=1136.125,396.861,-88.048,-176.849,11.356,149.493
C01483=1136.128,396.614,-88.010,-176.849,11.353,149.492
C01484=1136.132,396.367,-87.972,-176.849,11.351,149.492
C01485=1136.137,396.119,-87.934,-176.848,11.349,149.491
C01486=1136.140,395.873,-87.897,-176.849,11.347,149.490
C01487=1136.143,395.625,-87.859,-176.849,11.344,149.490
C01488=1136.148,395.378,-87.822,-176.848,11.342,149.489
C01489=1136.151,395.132,-87.785,-176.848,11.340,149.489
C01490=1136.155,394.884,-87.746,-176.849,11.338,149.488
C01491=1136.159,394.637,-87.708,-176.848,11.336,149.488
C01492=1136.163,394.390,-87.671,-176.849,11.334,149.487
C01493=1136.166,394.143,-87.634,-176.848,11.332,149.487
C01494=1136.170,393.896,-87.596,-176.848,11.330,149.486
C01495=1136.174,393.648,-87.558,-176.849,11.327,149.486
C01496=1136.178,393.401,-87.520,-176.849,11.326,149.485
C01497=1136.181,393.154,-87.483,-176.849,11.323,149.484
C01498=1136.185,392.908,-87.445,-176.849,11.321,149.484
C01499=1136.189,392.660,-87.408,-176.849,11.320,149.484
C01500=1136.192,392.413,-87.370,-176.850,11.317,149.483
C01501=1136.196,392.166,-87.332,-176.850,11.315,149.483
C01502=1136.200,391.919,-87.295,-176.850,11.314,149.482
C01503=1136.204,391.671,-87.257,-176.850,11.312,149.482
C01504=1136.207,391.425,-87.219,-176.851,11.310,149.482
C01505=1136.211,391.177,-87.182,-176.851,11.308,149.481
C01506=1136.215,390.930,-87.145,-176.851,11.306,149.481
C01507=1136.218,390.683,-87.107,-176.852,11.305,149.480
C01508=1136.223,390.436,-87.069,-176.852,11.303,149.480
C01509=1136.227,390.189,-87.032,-176.853,11.300,149.480
C01510=1136.229,389.976,-87.000,-176.853,11.299,149.479
C01511=1136.232,389.763,-86.967,-176.853,11.298,149.479
C01512=1136.235,389.550,-86.935,-176.854,11.296,149.479
C01513=1136.239,389.337,-86.903,-176.854,11.295,149.478
C01514=1136.242,389.124,-86.870,-176.855,11.293,149.478
C01515=1136.246,388.911,-86.838,-176.855,11.292,149.478
C01516=1136.248,388.698,-86.805,-176.855,11.291,149.478
C01517=1136.252,388.486,-86.774,-176.856,11.289,149.477
C01518=1136.255,388.239,-86.736,-176.856,11.288,149.477
C01519=1136.259,387.992,-86.698,-176.857,11.286,149.477
C01520=1136.263,387.744,-86.661,-176.858,11.284,149.477
C01521=1136.267,387.497,-86.623,-176.858,11.283,149.476
C01522=1136.271,387.250,-86.586,-176.859,11.281,149.476
C01523=1136.275,387.003,-86.548,-176.859,11.280,149.476
C01524=1136.278,386.756,-86.510,-176.860,11.278,149.476
C01525=1136.282,386.509,-86.473,-176.861,11.276,149.475
C01526=1136.285,386.261,-86.436,-176.861,11.275,149.475
C01527=1136.289,386.014,-86.399,-176.862,11.273,149.475
C01528=1136.293,385.768,-86.361,-176.863,11.271,149.475
C01529=1136.296,385.520,-86.324,-176.863,11.270,149.474
C01530=1136.300,385.273,-86.286,-176.865,11.269,149.474
C01531=1136.303,385.026,-86.248,-176.866,11.267,149.474
C01532=1136.308,384.778,-86.211,-176.866,11.266,149.474
C01533=1136.312,384.532,-86.173,-176.867,11.264,149.474
C01534=1136.315,384.284,-86.136,-176.868,11.263,149.474
C01535=1136.319,384.037,-86.099,-176.869,11.261,149.473
C01536=1136.323,383.789,-86.061,-176.870,11.260,149.473
C01537=1136.327,383.543,-86.024,-176.871,11.258,149.473
C01538=1136.331,383.296,-85.987,-176.872,11.257,149.473
C01539=1136.334,383.048,-85.949,-176.875,11.255,149.473
C01540=1136.338,382.801,-85.912,-176.877,11.253,149.473
C01541=1136.341,382.554,-85.874,-176.880,11.250,149.473
C01542=1136.345,382.307,-85.837,-176.882,11.248,149.473
C01543=1136.349,382.060,-85.800,-176.884,11.246,149.473
C01544=1136.353,381.812,-85.762,-176.887,11.243,149.473
C01545=1136.357,381.565,-85.726,-176.889,11.241,149.474
C01546=1136.360,381.319,-85.688,-176.892,11.239,149.474
C01547=1136.364,381.071,-85.651,-176.895,11.236,149.474
C01548=1136.368,380.824,-85.613,-176.897,11.234,149.474
C01549=1136.372,380.577,-85.576,-176.899,11.232,149.474
C01550=1136.375,380.329,-85.539,-176.902,11.230,149.474
C01551=1136.379,380.082,-85.502,-176.905,11.228,149.474
C01552=1136.383,379.835,-85.465,-176.907,11.225,149.474
C01553=1136.387,379.587,-85.427,-176.910,11.223,149.474
C01554=1136.390,379.341,-85.390,-176.913,11.221,149.474
C01555=1136.395,379.094,-85.353,-176.915,11.219,149.474
C01556=1136.398,378.846,-85.316,-176.918,11.216,149.474
C01557=1136.402,378.599,-85.278,-176.920,11.214,149.474
C01558=1136.405,378.352,-85.242,-176.923,11.212,149.475
C01559=1136.409,378.105,-85.205,-176.926,11.210,149.475
C01560=1136.413,377.857,-85.168,-176.928,11.208,149.475
C01561=1136.417,377.611,-85.130,-176.931,11.205,149.475
C01562=1136.421,377.363,-85.093,-176.933,11.203,149.475
C01563=1136.425,377.116,-85.057,-176.937,11.201,149.475
C01564=1136.428,376.868,-85.019,-176.939,11.199,149.475
C01565=1136.432,376.621,-84.983,-176.942,11.196,149.475
C01566=1136.435,376.409,-84.951,-176.944,11.195,149.476
C01567=1136.438,376.195,-84.918,-176.946,11.193,149.476
C01568=1136.442,375.982,-84.886,-176.949,11.191,149.476
C01569=1136.445,375.770,-84.855,-176.951,11.189,149.476
C01570=1136.448,375.556,-84.823,-176.953,11.187,149.476
C01571=1136.451,375.344,-84.792,-176.956,11.185,149.476
C01572=1136.455,375.131,-84.760,-176.958,11.183,149.476
C01573=1136.458,374.918,-84.729,-176.961,11.181,149.476
C01574=1136.462,374.670,-84.691,-176.964,11.179,149.477
C01575=1136.465,374.423,-84.654,-176.967,11.177,149.477
C01576=1136.470,374.176,-84.617,-176.970,11.174,149.477
C01577=1136.474,373.929,-84.580,-176.973,11.172,149.477
C01578=1136.476,373.681,-84.543,-176.976,11.170,149.477
C01579=1136.480,373.434,-84.507,-176.978,11.167,149.477
C01580=1136.485,373.187,-84.470,-176.981,11.166,149.478
C01581=1136.489,372.940,-84.433,-176.984,11.163,149.478
C01582=1136.492,372.693,-84.397,-176.987,11.161,149.478
C01583=1136.495,372.445,-84.359,-176.990,11.159,149.478
C01584=1136.500,372.198,-84.322,-176.993,11.157,149.478
C01585=1136.503,371.950,-84.287,-176.996,11.155,149.478
C01586=1136.507,371.703,-84.250,-176.999,11.152,149.478
C01587=1136.511,371.456,-84.213,-177.001,11.150,149.479
C01588=1136.515,371.209,-84.177,-177.005,11.148,149.479
C01589=1136.518,370.961,-84.140,-177.008,11.145,149.479
C01590=1136.522,370.714,-84.103,-177.011,11.143,149.479
C01591=1136.526,370.467,-84.067,-177.014,11.141,149.480
C01592=1136.530,370.220,-84.030,-177.017,11.139,149.480
C01593=1136.534,369.972,-83.994,-177.020,11.136,149.480
C01594=1136.538,369.725,-83.957,-177.023,11.134,149.480
C01595=1136.542,369.478,-83.920,-177.026,11.132,149.480
C01596=1136.546,369.231,-83.884,-177.029,11.130,149.481
C01597=1136.549,368.983,-83.847,-177.032,11.127,149.481
C01598=1136.553,368.736,-83.811,-177.036,11.125,149.481
C01599=1136.556,368.489,-83.775,-177.038,11.123,149.481
C01600=1136.560,368.241,-83.738,-177.041,11.121,149.481
C01601=1136.564,367.994,-83.701,-177.045,11.118,149.482
C01602=1136.568,367.747,-83.665,-177.048,11.116,149.482
C01603=1136.572,367.500,-83.628,-177.051,11.114,149.482
C01604=1136.576,367.253,-83.592,-177.054,11.112,149.482
C01605=1136.580,367.005,-83.556,-177.057,11.109,149.482
C01606=1136.583,366.758,-83.520,-177.061,11.107,149.483
C01607=1136.587,366.511,-83.483,-177.063,11.105,149.483
C01608=1136.592,366.263,-83.447,-177.067,11.102,149.483
C01609=1136.595,366.015,-83.410,-177.070,11.100,149.483
C01610=1136.599,365.768,-83.374,-177.073,11.097,149.484
C01611=1136.602,365.521,-83.338,-177.077,11.095,149.484
C01612=1136.606,365.274,-83.301,-177.080,11.093,149.484
C01613=1136.610,365.026,-83.265,-177.083,11.091,149.484
C01614=1136.613,364.779,-83.229,-177.086,11.089,149.485
C01615=1136.618,364.531,-83.193,-177.090,11.086,149.485
C01616=1136.621,364.284,-83.157,-177.093,11.084,149.485
C01617=1136.626,364.037,-83.121,-177.096,11.081,149.485
C01618=1136.629,363.790,-83.084,-177.099,11.079,149.486
C01619=1136.633,363.542,-83.048,-177.103,11.077,149.486
C01620=1136.637,363.295,-83.012,-177.106,11.074,149.486
C01621=1136.640,363.048,-82.976,-177.110,11.072,149.486
C01622=1136.644,362.835,-82.944,-177.112,11.070,149.487
C01623=1136.648,362.621,-82.914,-177.115,11.068,149.487
C01624=1136.651,362.408,-82.883,-177.118,11.066,149.487
C01625=1136.654,362.195,-82.852,-177.121,11.064,149.487
C01626=1136.657,361.982,-82.821,-177.124,11.061,149.487
C01627=1136.660,361.768,-82.789,-177.127,11.060,149.488
C01628=1136.664,361.555,-82.759,-177.129,11.058,149.488
C01629=1136.667,361.343,-82.727,-177.133,11.056,149.488
C01630=1136.671,361.095,-82.692,-177.136,11.053,149.488
C01631=1136.675,360.847,-82.656,-177.140,11.051,149.489
C01632=1136.678,360.600,-82.619,-177.143,11.048,149.489
C01633=1136.682,360.353,-82.584,-177.146,11.046,149.489
C01634=1136.686,360.106,-82.549,-177.150,11.044,149.489
C01635=1136.691,359.858,-82.513,-177.153,11.041,149.490
C01636=1136.694,359.611,-82.476,-177.157,11.039,149.490
C01637=1136.698,359.364,-82.441,-177.160,11.036,149.490
C01638=1136.702,359.116,-82.405,-177.163,11.034,149.490
C01639=1136.706,358.869,-82.369,-177.168,11.031,149.491
C01640=1136.709,358.621,-82.334,-177.171,11.029,149.491
C01641=1136.713,358.374,-82.298,-177.174,11.026,149.491
C01642=1136.716,358.127,-82.262,-177.178,11.024,149.492
C01643=1136.721,357.879,-82.226,-177.181,11.022,149.492
C01644=1136.725,357.632,-82.190,-177.184,11.019,149.492
C01645=1136.729,357.385,-82.155,-177.189,11.016,149.492
C01646=1136.732,357.137,-82.119,-177.192,11.014,149.493
C01647=1136.736,356.890,-82.084,-177.195,11.011,149.493
C01648=1136.740,356.642,-82.048,-177.199,11.009,149.493
C01649=1136.744,356.394,-82.012,-177.202,11.007,149.494
C01650=1136.748,356.147,-81.976,-177.206,11.003,149.494
C01651=1136.752,355.900,-81.941,-177.210,11.001,149.494
C01652=1136.756,355.652,-81.906,-177.213,10.999,149.494
C01653=1136.759,355.405,-81.870,-177.217,10.996,149.495
C01654=1136.763,355.157,-81.835,-177.221,10.993,149.495
C01655=1136.767,354.910,-81.799,-177.224,10.991,149.495
C01656=1136.772,354.663,-81.763,-177.228,10.988,149.495
C01657=1136.775,354.415,-81.728,-177.232,10.986,149.496
C01658=1136.779,354.168,-81.692,-177.235,10.983,149.496
C01659=1136.783,353.920,-81.657,-177.239,10.981,149.496
C01660=1136.787,353.672,-81.622,-177.243,10.978,149.497
C01661=1136.791,353.425,-81.587,-177.246,10.975,149.497
C01662=1136.795,353.178,-81.551,-177.250,10.972,149.497
C01663=1136.798,352.930,-81.516,-177.254,10.970,149.497
C01664=1136.802,352.683,-81.480,-177.257,10.967,149.498
C01665=1136.806,352.435,-81.446,-177.261,10.964,149.498
C01666=1136.810,352.188,-81.410,-177.265,10.962,149.498
C01667=1136.814,351.940,-81.374,-177.269,10.959,149.498
C01668=1136.818,351.693,-81.340,-177.272,10.956,149.499
C01669=1136.822,351.446,-81.304,-177.276,10.953,149.499
C01670=1136.826,351.198,-81.269,-177.280,10.951,149.499
C01671=1136.829,350.951,-81.233,-177.284,10.948,149.499
C01672=1136.834,350.703,-81.199,-177.287,10.946,149.500
C01673=1136.838,350.456,-81.163,-177.291,10.942,149.500
C01674=1136.842,350.208,-81.129,-177.295,10.940,149.500
C01675=1136.846,349.961,-81.093,-177.299,10.937,149.501
C01676=1136.849,349.714,-81.058,-177.302,10.935,149.501
C01677=1136.853,349.465,-81.024,-177.306,10.931,149.501
C01678=1136.859,349.107,-80.972,-177.311,10.928,149.501
C01679=1136.865,348.748,-80.922,-177.316,10.925,149.502
C01680=1136.870,348.389,-80.871,-177.321,10.921,149.502
C01681=1136.876,348.031,-80.820,-177.325,10.917,149.502
C01682=1136.880,347.782,-80.785,-177.328,10.915,149.503
C01683=1136.884,347.535,-80.751,-177.332,10.912,149.503
C01684=1136.888,347.288,-80.715,-177.335,10.910,149.503
C01685=1136.891,347.040,-80.681,-177.338,10.907,149.503
C01686=1136.895,346.793,-80.646,-177.342,10.905,149.503
C01687=1136.899,346.545,-80.611,-177.345,10.902,149.504
C01688=1136.904,346.297,-80.577,-177.348,10.900,149.504
C01689=1136.908,346.050,-80.541,-177.352,10.897,149.504
C01690=1136.911,345.802,-80.507,-177.355,10.895,149.504
C01691=1136.915,345.555,-80.472,-177.358,10.892,149.504
C01692=1136.919,345.307,-80.437,-177.361,10.890,149.505
C01693=1136.924,345.060,-80.402,-177.365,10.887,149.505
C01694=1136.927,344.812,-80.368,-177.368,10.885,149.505
C01695=1136.931,344.565,-80.333,-177.371,10.882,149.505
C01696=1136.935,344.317,-80.298,-177.374,10.880,149.506
C01697=1136.939,344.070,-80.264,-177.378,10.877,149.506
C01698=1136.943,343.822,-80.229,-177.381,10.875,149.506
C01699=1136.947,343.575,-80.194,-177.384,10.872,149.506
C01700=1136.950,343.327,-80.160,-177.387,10.870,149.506
C01701=1136.955,343.080,-80.126,-177.391,10.867,149.507
C01702=1136.959,342.832,-80.091,-177.394,10.865,149.507
C01703=1136.963,342.584,-80.057,-177.397,10.862,149.507
C01704=1136.967,342.336,-80.022,-177.401,10.860,149.507
C01705=1136.971,342.090,-79.987,-177.403,10.857,149.507
C01706=1136.974,341.842,-79.953,-177.407,10.855,149.508
C01707=1136.979,341.594,-79.918,-177.410,10.852,149.508
C01708=1136.983,341.346,-79.883,-177.413,10.850,149.508
C01709=1136.987,341.099,-79.849,-177.417,10.847,149.508
C01710=1136.991,340.851,-79.815,-177.420,10.845,149.508
C01711=1136.994,340.604,-79.781,-177.423,10.842,149.509
C01712=1136.998,340.356,-79.746,-177.426,10.840,149.509
C01713=1137.003,340.108,-79.711,-177.430,10.837,149.509
C01714=1137.006,339.861,-79.677,-177.433,10.835,149.509
C01715=1137.011,339.613,-79.643,-177.436,10.832,149.509
C01716=1137.014,339.365,-79.609,-177.439,10.829,149.510
C01717=1137.019,339.118,-79.574,-177.443,10.827,149.510
C01718=1137.038,337.896,-79.405,-176.637,9.259,148.896
C01719=1137.044,337.489,-79.349,-176.641,9.253,148.895
C01720=1137.049,337.242,-79.316,-176.644,9.249,148.895
C01721=1137.053,336.994,-79.281,-176.647,9.245,148.895
C01722=1137.056,336.746,-79.247,-176.649,9.241,148.895
C01723=1137.061,336.499,-79.214,-176.652,9.237,148.894
C01724=1137.064,336.251,-79.179,-176.655,9.233,148.894
C01725=1137.069,336.003,-79.146,-176.657,9.230,148.894
C01726=1137.072,335.756,-79.112,-176.660,9.225,148.893
C01727=1137.077,335.508,-79.079,-176.662,9.221,148.893
C01728=1137.081,335.260,-79.044,-176.665,9.218,148.893
C01729=1137.085,335.012,-79.011,-176.667,9.214,148.892
C01730=1137.089,334.765,-78.977,-176.670,9.210,148.892
C01731=1137.093,334.517,-78.944,-176.673,9.206,148.892
C01732=1137.096,334.269,-78.911,-176.675,9.202,148.891
C01733=1137.100,334.022,-78.877,-176.677,9.199,148.891
C01734=1137.105,333.774,-78.843,-176.680,9.195,148.891
C01735=1137.109,333.527,-78.809,-176.683,9.190,148.891
C01736=1137.112,333.278,-78.776,-176.685,9.187,148.890
C01737=1137.116,333.030,-78.743,-176.688,9.183,148.890
C01738=1137.120,332.783,-78.709,-176.691,9.179,148.890
C01739=1137.124,332.536,-78.676,-176.693,9.175,148.890
C01740=1137.129,332.288,-78.642,-176.696,9.171,148.889
C01741=1137.132,332.040,-78.608,-176.698,9.168,148.889
C01742=1137.137,331.792,-78.574,-176.701,9.164,148.889
C01743=1137.141,331.544,-78.541,-176.704,9.160,148.888
C01744=1137.145,331.297,-78.508,-176.706,9.156,148.888
C01745=1137.149,331.049,-78.475,-176.709,9.152,148.888
C01746=1137.153,330.802,-78.441,-176.711,9.149,148.888
C01747=1137.157,330.554,-78.408,-176.714,9.145,148.887
C01748=1137.161,330.306,-78.374,-176.717,9.140,148.887
C01749=1137.165,330.058,-78.341,-176.719,9.137,148.887
C01750=1137.169,329.810,-78.308,-176.722,9.133,148.887
C01751=1137.173,329.563,-78.274,-176.725,9.129,148.886
C01752=1137.177,329.315,-78.241,-176.727,9.126,148.886
C01753=1137.181,329.068,-78.208,-176.730,9.121,148.886
C01754=1137.185,328.820,-78.175,-176.732,9.118,148.885
C01755=1137.189,328.572,-78.142,-176.735,9.114,148.885
C01756=1137.193,328.324,-78.108,-176.738,9.110,148.885
C01757=1137.197,328.076,-78.075,-176.740,9.107,148.885
C01758=1137.201,327.828,-78.042,-176.743,9.102,148.885
C01759=1137.205,327.581,-78.009,-176.745,9.099,148.884
C01760=1137.209,327.333,-77.975,-176.748,9.095,148.884
C01761=1137.213,327.085,-77.942,-176.750,9.092,148.884
C01762=1137.218,326.837,-77.909,-176.753,9.087,148.884
C01763=1137.222,326.590,-77.876,-176.756,9.083,148.883
C01764=1137.226,326.342,-77.843,-176.758,9.080,148.883
C01765=1137.230,326.094,-77.810,-176.761,9.076,148.883
C01766=1137.233,325.847,-77.777,-176.763,9.072,148.883
C01767=1137.238,325.599,-77.744,-176.766,9.068,148.882
C01768=1137.242,325.351,-77.711,-176.769,9.064,148.882
C01769=1137.246,325.103,-77.678,-176.771,9.061,148.882
C01770=1137.250,324.855,-77.645,-176.774,9.057,148.882
C01771=1137.254,324.607,-77.612,-176.776,9.053,148.881
C01772=1137.259,324.360,-77.579,-176.779,9.049,148.881
C01773=1137.262,324.112,-77.546,-176.782,9.046,148.881
C01774=1137.266,323.865,-77.513,-176.785,9.042,148.881
C01775=1137.271,323.616,-77.481,-176.787,9.039,148.880
C01776=1137.275,323.368,-77.448,-176.790,9.035,148.880
C01777=1137.278,323.121,-77.415,-176.793,9.031,148.880
C01778=1137.282,322.873,-77.382,-176.795,9.027,148.880
C01779=1137.287,322.625,-77.349,-176.798,9.023,148.879
C01780=1137.291,322.377,-77.316,-176.800,9.020,148.879
C01781=1137.294,322.130,-77.284,-176.803,9.016,148.879
C01782=1137.299,321.881,-77.251,-176.805,9.012,148.879
C01783=1137.303,321.634,-77.218,-176.808,9.008,148.879
C01784=1137.306,321.386,-77.185,-176.810,9.005,148.878
C01785=1137.311,321.138,-77.153,-176.813,9.001,148.878
C01786=1137.315,320.890,-77.120,-176.816,8.997,148.878
C01787=1137.319,320.643,-77.087,-176.819,8.994,148.878
C01788=1137.323,320.394,-77.055,-176.822,8.990,148.877
C01789=1137.327,320.147,-77.022,-176.824,8.986,148.877
C01790=1137.330,319.899,-76.990,-176.827,8.982,148.877
C01791=1137.335,319.651,-76.957,-176.829,8.979,148.877
C01792=1137.339,319.403,-76.924,-176.832,8.975,148.877
C01793=1137.342,319.155,-76.892,-176.835,8.972,148.876
C01794=1137.347,318.908,-76.860,-176.837,8.967,148.876
C01795=1137.352,318.660,-76.827,-176.839,8.964,148.876
C01796=1137.355,318.412,-76.795,-176.842,8.960,148.876
C01797=1137.359,318.164,-76.762,-176.845,8.957,148.875
C01798=1137.363,317.916,-76.730,-176.848,8.953,148.875
C01799=1137.367,317.668,-76.697,-176.850,8.949,148.875
C01800=1137.371,317.420,-76.665,-176.853,8.945,148.875
